// NeuroPLC — Auto-generated IEC 61131-3 SCL (DB+FB Mode)
// Graph: mlp | Target: S71500DBBackend
// Work memory: 1500KB | LUT points: 0
// Nodes: 8 | Ops: {'matmul': 4, 'standard_act': 2, 'softmax': 1, 'argmax': 1}
// Parameters in DB "NeuroPLC_MLP_Weights", inference in FB.

FUNCTION_BLOCK "NeuroPLC_Inference"
{ S7_Optimized_Access := 'FALSE' }
VERSION : 0.1

VAR_INPUT
    features : ARRAY[0..27] OF REAL;  // 28-D feature vector
END_VAR

VAR_OUTPUT
    fault_class : INT;  // 0=Normal, 1=InnerRace, 2=Ball, 3=OuterRace
    confidence : REAL;  // max softmax probability
END_VAR

VAR
    // ── Inference temporaries ──
        v1 : ARRAY[0..31] OF REAL;  // matmul output
        v2 : ARRAY[0..31] OF REAL;  // relu output
        v3 : ARRAY[0..15] OF REAL;  // matmul output
        v4 : ARRAY[0..15] OF REAL;  // relu output
        v5 : ARRAY[0..3] OF REAL;  // matmul output
        v6 : ARRAY[0..3] OF REAL;  // softmax output

    // ── Temporary variables ──
    i, o, j, lo, hi, idx, base : INT;
    sum, max_val, t_val : REAL;
END_VAR

BEGIN
    // ═══ Inference forward pass ═══
    // Parameters loaded from DB "NeuroPLC_MLP_Weights" (start values = data, not code)

        // Input: features[0..27]

        // MatMul: fc0
        v1[0] := "NeuroPLC_MLP_Weights".b1[0] + "NeuroPLC_MLP_Weights".w0[0] * features[0] + "NeuroPLC_MLP_Weights".w0[1] * features[1] + "NeuroPLC_MLP_Weights".w0[2] * features[2] + "NeuroPLC_MLP_Weights".w0[3] * features[3] + "NeuroPLC_MLP_Weights".w0[4] * features[4] + "NeuroPLC_MLP_Weights".w0[5] * features[5] + "NeuroPLC_MLP_Weights".w0[6] * features[6] + "NeuroPLC_MLP_Weights".w0[7] * features[7] + "NeuroPLC_MLP_Weights".w0[8] * features[8] + "NeuroPLC_MLP_Weights".w0[9] * features[9] + "NeuroPLC_MLP_Weights".w0[10] * features[10] + "NeuroPLC_MLP_Weights".w0[11] * features[11] + "NeuroPLC_MLP_Weights".w0[12] * features[12] + "NeuroPLC_MLP_Weights".w0[13] * features[13] + "NeuroPLC_MLP_Weights".w0[14] * features[14] + "NeuroPLC_MLP_Weights".w0[15] * features[15] + "NeuroPLC_MLP_Weights".w0[16] * features[16] + "NeuroPLC_MLP_Weights".w0[17] * features[17] + "NeuroPLC_MLP_Weights".w0[18] * features[18] + "NeuroPLC_MLP_Weights".w0[19] * features[19] + "NeuroPLC_MLP_Weights".w0[20] * features[20] + "NeuroPLC_MLP_Weights".w0[21] * features[21] + "NeuroPLC_MLP_Weights".w0[22] * features[22] + "NeuroPLC_MLP_Weights".w0[23] * features[23] + "NeuroPLC_MLP_Weights".w0[24] * features[24] + "NeuroPLC_MLP_Weights".w0[25] * features[25] + "NeuroPLC_MLP_Weights".w0[26] * features[26] + "NeuroPLC_MLP_Weights".w0[27] * features[27];
        v1[1] := "NeuroPLC_MLP_Weights".b1[1] + "NeuroPLC_MLP_Weights".w0[28] * features[0] + "NeuroPLC_MLP_Weights".w0[29] * features[1] + "NeuroPLC_MLP_Weights".w0[30] * features[2] + "NeuroPLC_MLP_Weights".w0[31] * features[3] + "NeuroPLC_MLP_Weights".w0[32] * features[4] + "NeuroPLC_MLP_Weights".w0[33] * features[5] + "NeuroPLC_MLP_Weights".w0[34] * features[6] + "NeuroPLC_MLP_Weights".w0[35] * features[7] + "NeuroPLC_MLP_Weights".w0[36] * features[8] + "NeuroPLC_MLP_Weights".w0[37] * features[9] + "NeuroPLC_MLP_Weights".w0[38] * features[10] + "NeuroPLC_MLP_Weights".w0[39] * features[11] + "NeuroPLC_MLP_Weights".w0[40] * features[12] + "NeuroPLC_MLP_Weights".w0[41] * features[13] + "NeuroPLC_MLP_Weights".w0[42] * features[14] + "NeuroPLC_MLP_Weights".w0[43] * features[15] + "NeuroPLC_MLP_Weights".w0[44] * features[16] + "NeuroPLC_MLP_Weights".w0[45] * features[17] + "NeuroPLC_MLP_Weights".w0[46] * features[18] + "NeuroPLC_MLP_Weights".w0[47] * features[19] + "NeuroPLC_MLP_Weights".w0[48] * features[20] + "NeuroPLC_MLP_Weights".w0[49] * features[21] + "NeuroPLC_MLP_Weights".w0[50] * features[22] + "NeuroPLC_MLP_Weights".w0[51] * features[23] + "NeuroPLC_MLP_Weights".w0[52] * features[24] + "NeuroPLC_MLP_Weights".w0[53] * features[25] + "NeuroPLC_MLP_Weights".w0[54] * features[26] + "NeuroPLC_MLP_Weights".w0[55] * features[27];
        v1[2] := "NeuroPLC_MLP_Weights".b1[2] + "NeuroPLC_MLP_Weights".w0[56] * features[0] + "NeuroPLC_MLP_Weights".w0[57] * features[1] + "NeuroPLC_MLP_Weights".w0[58] * features[2] + "NeuroPLC_MLP_Weights".w0[59] * features[3] + "NeuroPLC_MLP_Weights".w0[60] * features[4] + "NeuroPLC_MLP_Weights".w0[61] * features[5] + "NeuroPLC_MLP_Weights".w0[62] * features[6] + "NeuroPLC_MLP_Weights".w0[63] * features[7] + "NeuroPLC_MLP_Weights".w0[64] * features[8] + "NeuroPLC_MLP_Weights".w0[65] * features[9] + "NeuroPLC_MLP_Weights".w0[66] * features[10] + "NeuroPLC_MLP_Weights".w0[67] * features[11] + "NeuroPLC_MLP_Weights".w0[68] * features[12] + "NeuroPLC_MLP_Weights".w0[69] * features[13] + "NeuroPLC_MLP_Weights".w0[70] * features[14] + "NeuroPLC_MLP_Weights".w0[71] * features[15] + "NeuroPLC_MLP_Weights".w0[72] * features[16] + "NeuroPLC_MLP_Weights".w0[73] * features[17] + "NeuroPLC_MLP_Weights".w0[74] * features[18] + "NeuroPLC_MLP_Weights".w0[75] * features[19] + "NeuroPLC_MLP_Weights".w0[76] * features[20] + "NeuroPLC_MLP_Weights".w0[77] * features[21] + "NeuroPLC_MLP_Weights".w0[78] * features[22] + "NeuroPLC_MLP_Weights".w0[79] * features[23] + "NeuroPLC_MLP_Weights".w0[80] * features[24] + "NeuroPLC_MLP_Weights".w0[81] * features[25] + "NeuroPLC_MLP_Weights".w0[82] * features[26] + "NeuroPLC_MLP_Weights".w0[83] * features[27];
        v1[3] := "NeuroPLC_MLP_Weights".b1[3] + "NeuroPLC_MLP_Weights".w0[84] * features[0] + "NeuroPLC_MLP_Weights".w0[85] * features[1] + "NeuroPLC_MLP_Weights".w0[86] * features[2] + "NeuroPLC_MLP_Weights".w0[87] * features[3] + "NeuroPLC_MLP_Weights".w0[88] * features[4] + "NeuroPLC_MLP_Weights".w0[89] * features[5] + "NeuroPLC_MLP_Weights".w0[90] * features[6] + "NeuroPLC_MLP_Weights".w0[91] * features[7] + "NeuroPLC_MLP_Weights".w0[92] * features[8] + "NeuroPLC_MLP_Weights".w0[93] * features[9] + "NeuroPLC_MLP_Weights".w0[94] * features[10] + "NeuroPLC_MLP_Weights".w0[95] * features[11] + "NeuroPLC_MLP_Weights".w0[96] * features[12] + "NeuroPLC_MLP_Weights".w0[97] * features[13] + "NeuroPLC_MLP_Weights".w0[98] * features[14] + "NeuroPLC_MLP_Weights".w0[99] * features[15] + "NeuroPLC_MLP_Weights".w0[100] * features[16] + "NeuroPLC_MLP_Weights".w0[101] * features[17] + "NeuroPLC_MLP_Weights".w0[102] * features[18] + "NeuroPLC_MLP_Weights".w0[103] * features[19] + "NeuroPLC_MLP_Weights".w0[104] * features[20] + "NeuroPLC_MLP_Weights".w0[105] * features[21] + "NeuroPLC_MLP_Weights".w0[106] * features[22] + "NeuroPLC_MLP_Weights".w0[107] * features[23] + "NeuroPLC_MLP_Weights".w0[108] * features[24] + "NeuroPLC_MLP_Weights".w0[109] * features[25] + "NeuroPLC_MLP_Weights".w0[110] * features[26] + "NeuroPLC_MLP_Weights".w0[111] * features[27];
        v1[4] := "NeuroPLC_MLP_Weights".b1[4] + "NeuroPLC_MLP_Weights".w0[112] * features[0] + "NeuroPLC_MLP_Weights".w0[113] * features[1] + "NeuroPLC_MLP_Weights".w0[114] * features[2] + "NeuroPLC_MLP_Weights".w0[115] * features[3] + "NeuroPLC_MLP_Weights".w0[116] * features[4] + "NeuroPLC_MLP_Weights".w0[117] * features[5] + "NeuroPLC_MLP_Weights".w0[118] * features[6] + "NeuroPLC_MLP_Weights".w0[119] * features[7] + "NeuroPLC_MLP_Weights".w0[120] * features[8] + "NeuroPLC_MLP_Weights".w0[121] * features[9] + "NeuroPLC_MLP_Weights".w0[122] * features[10] + "NeuroPLC_MLP_Weights".w0[123] * features[11] + "NeuroPLC_MLP_Weights".w0[124] * features[12] + "NeuroPLC_MLP_Weights".w0[125] * features[13] + "NeuroPLC_MLP_Weights".w0[126] * features[14] + "NeuroPLC_MLP_Weights".w0[127] * features[15] + "NeuroPLC_MLP_Weights".w0[128] * features[16] + "NeuroPLC_MLP_Weights".w0[129] * features[17] + "NeuroPLC_MLP_Weights".w0[130] * features[18] + "NeuroPLC_MLP_Weights".w0[131] * features[19] + "NeuroPLC_MLP_Weights".w0[132] * features[20] + "NeuroPLC_MLP_Weights".w0[133] * features[21] + "NeuroPLC_MLP_Weights".w0[134] * features[22] + "NeuroPLC_MLP_Weights".w0[135] * features[23] + "NeuroPLC_MLP_Weights".w0[136] * features[24] + "NeuroPLC_MLP_Weights".w0[137] * features[25] + "NeuroPLC_MLP_Weights".w0[138] * features[26] + "NeuroPLC_MLP_Weights".w0[139] * features[27];
        v1[5] := "NeuroPLC_MLP_Weights".b1[5] + "NeuroPLC_MLP_Weights".w0[140] * features[0] + "NeuroPLC_MLP_Weights".w0[141] * features[1] + "NeuroPLC_MLP_Weights".w0[142] * features[2] + "NeuroPLC_MLP_Weights".w0[143] * features[3] + "NeuroPLC_MLP_Weights".w0[144] * features[4] + "NeuroPLC_MLP_Weights".w0[145] * features[5] + "NeuroPLC_MLP_Weights".w0[146] * features[6] + "NeuroPLC_MLP_Weights".w0[147] * features[7] + "NeuroPLC_MLP_Weights".w0[148] * features[8] + "NeuroPLC_MLP_Weights".w0[149] * features[9] + "NeuroPLC_MLP_Weights".w0[150] * features[10] + "NeuroPLC_MLP_Weights".w0[151] * features[11] + "NeuroPLC_MLP_Weights".w0[152] * features[12] + "NeuroPLC_MLP_Weights".w0[153] * features[13] + "NeuroPLC_MLP_Weights".w0[154] * features[14] + "NeuroPLC_MLP_Weights".w0[155] * features[15] + "NeuroPLC_MLP_Weights".w0[156] * features[16] + "NeuroPLC_MLP_Weights".w0[157] * features[17] + "NeuroPLC_MLP_Weights".w0[158] * features[18] + "NeuroPLC_MLP_Weights".w0[159] * features[19] + "NeuroPLC_MLP_Weights".w0[160] * features[20] + "NeuroPLC_MLP_Weights".w0[161] * features[21] + "NeuroPLC_MLP_Weights".w0[162] * features[22] + "NeuroPLC_MLP_Weights".w0[163] * features[23] + "NeuroPLC_MLP_Weights".w0[164] * features[24] + "NeuroPLC_MLP_Weights".w0[165] * features[25] + "NeuroPLC_MLP_Weights".w0[166] * features[26] + "NeuroPLC_MLP_Weights".w0[167] * features[27];
        v1[6] := "NeuroPLC_MLP_Weights".b1[6] + "NeuroPLC_MLP_Weights".w0[168] * features[0] + "NeuroPLC_MLP_Weights".w0[169] * features[1] + "NeuroPLC_MLP_Weights".w0[170] * features[2] + "NeuroPLC_MLP_Weights".w0[171] * features[3] + "NeuroPLC_MLP_Weights".w0[172] * features[4] + "NeuroPLC_MLP_Weights".w0[173] * features[5] + "NeuroPLC_MLP_Weights".w0[174] * features[6] + "NeuroPLC_MLP_Weights".w0[175] * features[7] + "NeuroPLC_MLP_Weights".w0[176] * features[8] + "NeuroPLC_MLP_Weights".w0[177] * features[9] + "NeuroPLC_MLP_Weights".w0[178] * features[10] + "NeuroPLC_MLP_Weights".w0[179] * features[11] + "NeuroPLC_MLP_Weights".w0[180] * features[12] + "NeuroPLC_MLP_Weights".w0[181] * features[13] + "NeuroPLC_MLP_Weights".w0[182] * features[14] + "NeuroPLC_MLP_Weights".w0[183] * features[15] + "NeuroPLC_MLP_Weights".w0[184] * features[16] + "NeuroPLC_MLP_Weights".w0[185] * features[17] + "NeuroPLC_MLP_Weights".w0[186] * features[18] + "NeuroPLC_MLP_Weights".w0[187] * features[19] + "NeuroPLC_MLP_Weights".w0[188] * features[20] + "NeuroPLC_MLP_Weights".w0[189] * features[21] + "NeuroPLC_MLP_Weights".w0[190] * features[22] + "NeuroPLC_MLP_Weights".w0[191] * features[23] + "NeuroPLC_MLP_Weights".w0[192] * features[24] + "NeuroPLC_MLP_Weights".w0[193] * features[25] + "NeuroPLC_MLP_Weights".w0[194] * features[26] + "NeuroPLC_MLP_Weights".w0[195] * features[27];
        v1[7] := "NeuroPLC_MLP_Weights".b1[7] + "NeuroPLC_MLP_Weights".w0[196] * features[0] + "NeuroPLC_MLP_Weights".w0[197] * features[1] + "NeuroPLC_MLP_Weights".w0[198] * features[2] + "NeuroPLC_MLP_Weights".w0[199] * features[3] + "NeuroPLC_MLP_Weights".w0[200] * features[4] + "NeuroPLC_MLP_Weights".w0[201] * features[5] + "NeuroPLC_MLP_Weights".w0[202] * features[6] + "NeuroPLC_MLP_Weights".w0[203] * features[7] + "NeuroPLC_MLP_Weights".w0[204] * features[8] + "NeuroPLC_MLP_Weights".w0[205] * features[9] + "NeuroPLC_MLP_Weights".w0[206] * features[10] + "NeuroPLC_MLP_Weights".w0[207] * features[11] + "NeuroPLC_MLP_Weights".w0[208] * features[12] + "NeuroPLC_MLP_Weights".w0[209] * features[13] + "NeuroPLC_MLP_Weights".w0[210] * features[14] + "NeuroPLC_MLP_Weights".w0[211] * features[15] + "NeuroPLC_MLP_Weights".w0[212] * features[16] + "NeuroPLC_MLP_Weights".w0[213] * features[17] + "NeuroPLC_MLP_Weights".w0[214] * features[18] + "NeuroPLC_MLP_Weights".w0[215] * features[19] + "NeuroPLC_MLP_Weights".w0[216] * features[20] + "NeuroPLC_MLP_Weights".w0[217] * features[21] + "NeuroPLC_MLP_Weights".w0[218] * features[22] + "NeuroPLC_MLP_Weights".w0[219] * features[23] + "NeuroPLC_MLP_Weights".w0[220] * features[24] + "NeuroPLC_MLP_Weights".w0[221] * features[25] + "NeuroPLC_MLP_Weights".w0[222] * features[26] + "NeuroPLC_MLP_Weights".w0[223] * features[27];
        v1[8] := "NeuroPLC_MLP_Weights".b1[8] + "NeuroPLC_MLP_Weights".w0[224] * features[0] + "NeuroPLC_MLP_Weights".w0[225] * features[1] + "NeuroPLC_MLP_Weights".w0[226] * features[2] + "NeuroPLC_MLP_Weights".w0[227] * features[3] + "NeuroPLC_MLP_Weights".w0[228] * features[4] + "NeuroPLC_MLP_Weights".w0[229] * features[5] + "NeuroPLC_MLP_Weights".w0[230] * features[6] + "NeuroPLC_MLP_Weights".w0[231] * features[7] + "NeuroPLC_MLP_Weights".w0[232] * features[8] + "NeuroPLC_MLP_Weights".w0[233] * features[9] + "NeuroPLC_MLP_Weights".w0[234] * features[10] + "NeuroPLC_MLP_Weights".w0[235] * features[11] + "NeuroPLC_MLP_Weights".w0[236] * features[12] + "NeuroPLC_MLP_Weights".w0[237] * features[13] + "NeuroPLC_MLP_Weights".w0[238] * features[14] + "NeuroPLC_MLP_Weights".w0[239] * features[15] + "NeuroPLC_MLP_Weights".w0[240] * features[16] + "NeuroPLC_MLP_Weights".w0[241] * features[17] + "NeuroPLC_MLP_Weights".w0[242] * features[18] + "NeuroPLC_MLP_Weights".w0[243] * features[19] + "NeuroPLC_MLP_Weights".w0[244] * features[20] + "NeuroPLC_MLP_Weights".w0[245] * features[21] + "NeuroPLC_MLP_Weights".w0[246] * features[22] + "NeuroPLC_MLP_Weights".w0[247] * features[23] + "NeuroPLC_MLP_Weights".w0[248] * features[24] + "NeuroPLC_MLP_Weights".w0[249] * features[25] + "NeuroPLC_MLP_Weights".w0[250] * features[26] + "NeuroPLC_MLP_Weights".w0[251] * features[27];
        v1[9] := "NeuroPLC_MLP_Weights".b1[9] + "NeuroPLC_MLP_Weights".w0[252] * features[0] + "NeuroPLC_MLP_Weights".w0[253] * features[1] + "NeuroPLC_MLP_Weights".w0[254] * features[2] + "NeuroPLC_MLP_Weights".w0[255] * features[3] + "NeuroPLC_MLP_Weights".w0[256] * features[4] + "NeuroPLC_MLP_Weights".w0[257] * features[5] + "NeuroPLC_MLP_Weights".w0[258] * features[6] + "NeuroPLC_MLP_Weights".w0[259] * features[7] + "NeuroPLC_MLP_Weights".w0[260] * features[8] + "NeuroPLC_MLP_Weights".w0[261] * features[9] + "NeuroPLC_MLP_Weights".w0[262] * features[10] + "NeuroPLC_MLP_Weights".w0[263] * features[11] + "NeuroPLC_MLP_Weights".w0[264] * features[12] + "NeuroPLC_MLP_Weights".w0[265] * features[13] + "NeuroPLC_MLP_Weights".w0[266] * features[14] + "NeuroPLC_MLP_Weights".w0[267] * features[15] + "NeuroPLC_MLP_Weights".w0[268] * features[16] + "NeuroPLC_MLP_Weights".w0[269] * features[17] + "NeuroPLC_MLP_Weights".w0[270] * features[18] + "NeuroPLC_MLP_Weights".w0[271] * features[19] + "NeuroPLC_MLP_Weights".w0[272] * features[20] + "NeuroPLC_MLP_Weights".w0[273] * features[21] + "NeuroPLC_MLP_Weights".w0[274] * features[22] + "NeuroPLC_MLP_Weights".w0[275] * features[23] + "NeuroPLC_MLP_Weights".w0[276] * features[24] + "NeuroPLC_MLP_Weights".w0[277] * features[25] + "NeuroPLC_MLP_Weights".w0[278] * features[26] + "NeuroPLC_MLP_Weights".w0[279] * features[27];
        v1[10] := "NeuroPLC_MLP_Weights".b1[10] + "NeuroPLC_MLP_Weights".w0[280] * features[0] + "NeuroPLC_MLP_Weights".w0[281] * features[1] + "NeuroPLC_MLP_Weights".w0[282] * features[2] + "NeuroPLC_MLP_Weights".w0[283] * features[3] + "NeuroPLC_MLP_Weights".w0[284] * features[4] + "NeuroPLC_MLP_Weights".w0[285] * features[5] + "NeuroPLC_MLP_Weights".w0[286] * features[6] + "NeuroPLC_MLP_Weights".w0[287] * features[7] + "NeuroPLC_MLP_Weights".w0[288] * features[8] + "NeuroPLC_MLP_Weights".w0[289] * features[9] + "NeuroPLC_MLP_Weights".w0[290] * features[10] + "NeuroPLC_MLP_Weights".w0[291] * features[11] + "NeuroPLC_MLP_Weights".w0[292] * features[12] + "NeuroPLC_MLP_Weights".w0[293] * features[13] + "NeuroPLC_MLP_Weights".w0[294] * features[14] + "NeuroPLC_MLP_Weights".w0[295] * features[15] + "NeuroPLC_MLP_Weights".w0[296] * features[16] + "NeuroPLC_MLP_Weights".w0[297] * features[17] + "NeuroPLC_MLP_Weights".w0[298] * features[18] + "NeuroPLC_MLP_Weights".w0[299] * features[19] + "NeuroPLC_MLP_Weights".w0[300] * features[20] + "NeuroPLC_MLP_Weights".w0[301] * features[21] + "NeuroPLC_MLP_Weights".w0[302] * features[22] + "NeuroPLC_MLP_Weights".w0[303] * features[23] + "NeuroPLC_MLP_Weights".w0[304] * features[24] + "NeuroPLC_MLP_Weights".w0[305] * features[25] + "NeuroPLC_MLP_Weights".w0[306] * features[26] + "NeuroPLC_MLP_Weights".w0[307] * features[27];
        v1[11] := "NeuroPLC_MLP_Weights".b1[11] + "NeuroPLC_MLP_Weights".w0[308] * features[0] + "NeuroPLC_MLP_Weights".w0[309] * features[1] + "NeuroPLC_MLP_Weights".w0[310] * features[2] + "NeuroPLC_MLP_Weights".w0[311] * features[3] + "NeuroPLC_MLP_Weights".w0[312] * features[4] + "NeuroPLC_MLP_Weights".w0[313] * features[5] + "NeuroPLC_MLP_Weights".w0[314] * features[6] + "NeuroPLC_MLP_Weights".w0[315] * features[7] + "NeuroPLC_MLP_Weights".w0[316] * features[8] + "NeuroPLC_MLP_Weights".w0[317] * features[9] + "NeuroPLC_MLP_Weights".w0[318] * features[10] + "NeuroPLC_MLP_Weights".w0[319] * features[11] + "NeuroPLC_MLP_Weights".w0[320] * features[12] + "NeuroPLC_MLP_Weights".w0[321] * features[13] + "NeuroPLC_MLP_Weights".w0[322] * features[14] + "NeuroPLC_MLP_Weights".w0[323] * features[15] + "NeuroPLC_MLP_Weights".w0[324] * features[16] + "NeuroPLC_MLP_Weights".w0[325] * features[17] + "NeuroPLC_MLP_Weights".w0[326] * features[18] + "NeuroPLC_MLP_Weights".w0[327] * features[19] + "NeuroPLC_MLP_Weights".w0[328] * features[20] + "NeuroPLC_MLP_Weights".w0[329] * features[21] + "NeuroPLC_MLP_Weights".w0[330] * features[22] + "NeuroPLC_MLP_Weights".w0[331] * features[23] + "NeuroPLC_MLP_Weights".w0[332] * features[24] + "NeuroPLC_MLP_Weights".w0[333] * features[25] + "NeuroPLC_MLP_Weights".w0[334] * features[26] + "NeuroPLC_MLP_Weights".w0[335] * features[27];
        v1[12] := "NeuroPLC_MLP_Weights".b1[12] + "NeuroPLC_MLP_Weights".w0[336] * features[0] + "NeuroPLC_MLP_Weights".w0[337] * features[1] + "NeuroPLC_MLP_Weights".w0[338] * features[2] + "NeuroPLC_MLP_Weights".w0[339] * features[3] + "NeuroPLC_MLP_Weights".w0[340] * features[4] + "NeuroPLC_MLP_Weights".w0[341] * features[5] + "NeuroPLC_MLP_Weights".w0[342] * features[6] + "NeuroPLC_MLP_Weights".w0[343] * features[7] + "NeuroPLC_MLP_Weights".w0[344] * features[8] + "NeuroPLC_MLP_Weights".w0[345] * features[9] + "NeuroPLC_MLP_Weights".w0[346] * features[10] + "NeuroPLC_MLP_Weights".w0[347] * features[11] + "NeuroPLC_MLP_Weights".w0[348] * features[12] + "NeuroPLC_MLP_Weights".w0[349] * features[13] + "NeuroPLC_MLP_Weights".w0[350] * features[14] + "NeuroPLC_MLP_Weights".w0[351] * features[15] + "NeuroPLC_MLP_Weights".w0[352] * features[16] + "NeuroPLC_MLP_Weights".w0[353] * features[17] + "NeuroPLC_MLP_Weights".w0[354] * features[18] + "NeuroPLC_MLP_Weights".w0[355] * features[19] + "NeuroPLC_MLP_Weights".w0[356] * features[20] + "NeuroPLC_MLP_Weights".w0[357] * features[21] + "NeuroPLC_MLP_Weights".w0[358] * features[22] + "NeuroPLC_MLP_Weights".w0[359] * features[23] + "NeuroPLC_MLP_Weights".w0[360] * features[24] + "NeuroPLC_MLP_Weights".w0[361] * features[25] + "NeuroPLC_MLP_Weights".w0[362] * features[26] + "NeuroPLC_MLP_Weights".w0[363] * features[27];
        v1[13] := "NeuroPLC_MLP_Weights".b1[13] + "NeuroPLC_MLP_Weights".w0[364] * features[0] + "NeuroPLC_MLP_Weights".w0[365] * features[1] + "NeuroPLC_MLP_Weights".w0[366] * features[2] + "NeuroPLC_MLP_Weights".w0[367] * features[3] + "NeuroPLC_MLP_Weights".w0[368] * features[4] + "NeuroPLC_MLP_Weights".w0[369] * features[5] + "NeuroPLC_MLP_Weights".w0[370] * features[6] + "NeuroPLC_MLP_Weights".w0[371] * features[7] + "NeuroPLC_MLP_Weights".w0[372] * features[8] + "NeuroPLC_MLP_Weights".w0[373] * features[9] + "NeuroPLC_MLP_Weights".w0[374] * features[10] + "NeuroPLC_MLP_Weights".w0[375] * features[11] + "NeuroPLC_MLP_Weights".w0[376] * features[12] + "NeuroPLC_MLP_Weights".w0[377] * features[13] + "NeuroPLC_MLP_Weights".w0[378] * features[14] + "NeuroPLC_MLP_Weights".w0[379] * features[15] + "NeuroPLC_MLP_Weights".w0[380] * features[16] + "NeuroPLC_MLP_Weights".w0[381] * features[17] + "NeuroPLC_MLP_Weights".w0[382] * features[18] + "NeuroPLC_MLP_Weights".w0[383] * features[19] + "NeuroPLC_MLP_Weights".w0[384] * features[20] + "NeuroPLC_MLP_Weights".w0[385] * features[21] + "NeuroPLC_MLP_Weights".w0[386] * features[22] + "NeuroPLC_MLP_Weights".w0[387] * features[23] + "NeuroPLC_MLP_Weights".w0[388] * features[24] + "NeuroPLC_MLP_Weights".w0[389] * features[25] + "NeuroPLC_MLP_Weights".w0[390] * features[26] + "NeuroPLC_MLP_Weights".w0[391] * features[27];
        v1[14] := "NeuroPLC_MLP_Weights".b1[14] + "NeuroPLC_MLP_Weights".w0[392] * features[0] + "NeuroPLC_MLP_Weights".w0[393] * features[1] + "NeuroPLC_MLP_Weights".w0[394] * features[2] + "NeuroPLC_MLP_Weights".w0[395] * features[3] + "NeuroPLC_MLP_Weights".w0[396] * features[4] + "NeuroPLC_MLP_Weights".w0[397] * features[5] + "NeuroPLC_MLP_Weights".w0[398] * features[6] + "NeuroPLC_MLP_Weights".w0[399] * features[7] + "NeuroPLC_MLP_Weights".w0[400] * features[8] + "NeuroPLC_MLP_Weights".w0[401] * features[9] + "NeuroPLC_MLP_Weights".w0[402] * features[10] + "NeuroPLC_MLP_Weights".w0[403] * features[11] + "NeuroPLC_MLP_Weights".w0[404] * features[12] + "NeuroPLC_MLP_Weights".w0[405] * features[13] + "NeuroPLC_MLP_Weights".w0[406] * features[14] + "NeuroPLC_MLP_Weights".w0[407] * features[15] + "NeuroPLC_MLP_Weights".w0[408] * features[16] + "NeuroPLC_MLP_Weights".w0[409] * features[17] + "NeuroPLC_MLP_Weights".w0[410] * features[18] + "NeuroPLC_MLP_Weights".w0[411] * features[19] + "NeuroPLC_MLP_Weights".w0[412] * features[20] + "NeuroPLC_MLP_Weights".w0[413] * features[21] + "NeuroPLC_MLP_Weights".w0[414] * features[22] + "NeuroPLC_MLP_Weights".w0[415] * features[23] + "NeuroPLC_MLP_Weights".w0[416] * features[24] + "NeuroPLC_MLP_Weights".w0[417] * features[25] + "NeuroPLC_MLP_Weights".w0[418] * features[26] + "NeuroPLC_MLP_Weights".w0[419] * features[27];
        v1[15] := "NeuroPLC_MLP_Weights".b1[15] + "NeuroPLC_MLP_Weights".w0[420] * features[0] + "NeuroPLC_MLP_Weights".w0[421] * features[1] + "NeuroPLC_MLP_Weights".w0[422] * features[2] + "NeuroPLC_MLP_Weights".w0[423] * features[3] + "NeuroPLC_MLP_Weights".w0[424] * features[4] + "NeuroPLC_MLP_Weights".w0[425] * features[5] + "NeuroPLC_MLP_Weights".w0[426] * features[6] + "NeuroPLC_MLP_Weights".w0[427] * features[7] + "NeuroPLC_MLP_Weights".w0[428] * features[8] + "NeuroPLC_MLP_Weights".w0[429] * features[9] + "NeuroPLC_MLP_Weights".w0[430] * features[10] + "NeuroPLC_MLP_Weights".w0[431] * features[11] + "NeuroPLC_MLP_Weights".w0[432] * features[12] + "NeuroPLC_MLP_Weights".w0[433] * features[13] + "NeuroPLC_MLP_Weights".w0[434] * features[14] + "NeuroPLC_MLP_Weights".w0[435] * features[15] + "NeuroPLC_MLP_Weights".w0[436] * features[16] + "NeuroPLC_MLP_Weights".w0[437] * features[17] + "NeuroPLC_MLP_Weights".w0[438] * features[18] + "NeuroPLC_MLP_Weights".w0[439] * features[19] + "NeuroPLC_MLP_Weights".w0[440] * features[20] + "NeuroPLC_MLP_Weights".w0[441] * features[21] + "NeuroPLC_MLP_Weights".w0[442] * features[22] + "NeuroPLC_MLP_Weights".w0[443] * features[23] + "NeuroPLC_MLP_Weights".w0[444] * features[24] + "NeuroPLC_MLP_Weights".w0[445] * features[25] + "NeuroPLC_MLP_Weights".w0[446] * features[26] + "NeuroPLC_MLP_Weights".w0[447] * features[27];
        v1[16] := "NeuroPLC_MLP_Weights".b1[16] + "NeuroPLC_MLP_Weights".w0[448] * features[0] + "NeuroPLC_MLP_Weights".w0[449] * features[1] + "NeuroPLC_MLP_Weights".w0[450] * features[2] + "NeuroPLC_MLP_Weights".w0[451] * features[3] + "NeuroPLC_MLP_Weights".w0[452] * features[4] + "NeuroPLC_MLP_Weights".w0[453] * features[5] + "NeuroPLC_MLP_Weights".w0[454] * features[6] + "NeuroPLC_MLP_Weights".w0[455] * features[7] + "NeuroPLC_MLP_Weights".w0[456] * features[8] + "NeuroPLC_MLP_Weights".w0[457] * features[9] + "NeuroPLC_MLP_Weights".w0[458] * features[10] + "NeuroPLC_MLP_Weights".w0[459] * features[11] + "NeuroPLC_MLP_Weights".w0[460] * features[12] + "NeuroPLC_MLP_Weights".w0[461] * features[13] + "NeuroPLC_MLP_Weights".w0[462] * features[14] + "NeuroPLC_MLP_Weights".w0[463] * features[15] + "NeuroPLC_MLP_Weights".w0[464] * features[16] + "NeuroPLC_MLP_Weights".w0[465] * features[17] + "NeuroPLC_MLP_Weights".w0[466] * features[18] + "NeuroPLC_MLP_Weights".w0[467] * features[19] + "NeuroPLC_MLP_Weights".w0[468] * features[20] + "NeuroPLC_MLP_Weights".w0[469] * features[21] + "NeuroPLC_MLP_Weights".w0[470] * features[22] + "NeuroPLC_MLP_Weights".w0[471] * features[23] + "NeuroPLC_MLP_Weights".w0[472] * features[24] + "NeuroPLC_MLP_Weights".w0[473] * features[25] + "NeuroPLC_MLP_Weights".w0[474] * features[26] + "NeuroPLC_MLP_Weights".w0[475] * features[27];
        v1[17] := "NeuroPLC_MLP_Weights".b1[17] + "NeuroPLC_MLP_Weights".w0[476] * features[0] + "NeuroPLC_MLP_Weights".w0[477] * features[1] + "NeuroPLC_MLP_Weights".w0[478] * features[2] + "NeuroPLC_MLP_Weights".w0[479] * features[3] + "NeuroPLC_MLP_Weights".w0[480] * features[4] + "NeuroPLC_MLP_Weights".w0[481] * features[5] + "NeuroPLC_MLP_Weights".w0[482] * features[6] + "NeuroPLC_MLP_Weights".w0[483] * features[7] + "NeuroPLC_MLP_Weights".w0[484] * features[8] + "NeuroPLC_MLP_Weights".w0[485] * features[9] + "NeuroPLC_MLP_Weights".w0[486] * features[10] + "NeuroPLC_MLP_Weights".w0[487] * features[11] + "NeuroPLC_MLP_Weights".w0[488] * features[12] + "NeuroPLC_MLP_Weights".w0[489] * features[13] + "NeuroPLC_MLP_Weights".w0[490] * features[14] + "NeuroPLC_MLP_Weights".w0[491] * features[15] + "NeuroPLC_MLP_Weights".w0[492] * features[16] + "NeuroPLC_MLP_Weights".w0[493] * features[17] + "NeuroPLC_MLP_Weights".w0[494] * features[18] + "NeuroPLC_MLP_Weights".w0[495] * features[19] + "NeuroPLC_MLP_Weights".w0[496] * features[20] + "NeuroPLC_MLP_Weights".w0[497] * features[21] + "NeuroPLC_MLP_Weights".w0[498] * features[22] + "NeuroPLC_MLP_Weights".w0[499] * features[23] + "NeuroPLC_MLP_Weights".w0[500] * features[24] + "NeuroPLC_MLP_Weights".w0[501] * features[25] + "NeuroPLC_MLP_Weights".w0[502] * features[26] + "NeuroPLC_MLP_Weights".w0[503] * features[27];
        v1[18] := "NeuroPLC_MLP_Weights".b1[18] + "NeuroPLC_MLP_Weights".w0[504] * features[0] + "NeuroPLC_MLP_Weights".w0[505] * features[1] + "NeuroPLC_MLP_Weights".w0[506] * features[2] + "NeuroPLC_MLP_Weights".w0[507] * features[3] + "NeuroPLC_MLP_Weights".w0[508] * features[4] + "NeuroPLC_MLP_Weights".w0[509] * features[5] + "NeuroPLC_MLP_Weights".w0[510] * features[6] + "NeuroPLC_MLP_Weights".w0[511] * features[7] + "NeuroPLC_MLP_Weights".w0[512] * features[8] + "NeuroPLC_MLP_Weights".w0[513] * features[9] + "NeuroPLC_MLP_Weights".w0[514] * features[10] + "NeuroPLC_MLP_Weights".w0[515] * features[11] + "NeuroPLC_MLP_Weights".w0[516] * features[12] + "NeuroPLC_MLP_Weights".w0[517] * features[13] + "NeuroPLC_MLP_Weights".w0[518] * features[14] + "NeuroPLC_MLP_Weights".w0[519] * features[15] + "NeuroPLC_MLP_Weights".w0[520] * features[16] + "NeuroPLC_MLP_Weights".w0[521] * features[17] + "NeuroPLC_MLP_Weights".w0[522] * features[18] + "NeuroPLC_MLP_Weights".w0[523] * features[19] + "NeuroPLC_MLP_Weights".w0[524] * features[20] + "NeuroPLC_MLP_Weights".w0[525] * features[21] + "NeuroPLC_MLP_Weights".w0[526] * features[22] + "NeuroPLC_MLP_Weights".w0[527] * features[23] + "NeuroPLC_MLP_Weights".w0[528] * features[24] + "NeuroPLC_MLP_Weights".w0[529] * features[25] + "NeuroPLC_MLP_Weights".w0[530] * features[26] + "NeuroPLC_MLP_Weights".w0[531] * features[27];
        v1[19] := "NeuroPLC_MLP_Weights".b1[19] + "NeuroPLC_MLP_Weights".w0[532] * features[0] + "NeuroPLC_MLP_Weights".w0[533] * features[1] + "NeuroPLC_MLP_Weights".w0[534] * features[2] + "NeuroPLC_MLP_Weights".w0[535] * features[3] + "NeuroPLC_MLP_Weights".w0[536] * features[4] + "NeuroPLC_MLP_Weights".w0[537] * features[5] + "NeuroPLC_MLP_Weights".w0[538] * features[6] + "NeuroPLC_MLP_Weights".w0[539] * features[7] + "NeuroPLC_MLP_Weights".w0[540] * features[8] + "NeuroPLC_MLP_Weights".w0[541] * features[9] + "NeuroPLC_MLP_Weights".w0[542] * features[10] + "NeuroPLC_MLP_Weights".w0[543] * features[11] + "NeuroPLC_MLP_Weights".w0[544] * features[12] + "NeuroPLC_MLP_Weights".w0[545] * features[13] + "NeuroPLC_MLP_Weights".w0[546] * features[14] + "NeuroPLC_MLP_Weights".w0[547] * features[15] + "NeuroPLC_MLP_Weights".w0[548] * features[16] + "NeuroPLC_MLP_Weights".w0[549] * features[17] + "NeuroPLC_MLP_Weights".w0[550] * features[18] + "NeuroPLC_MLP_Weights".w0[551] * features[19] + "NeuroPLC_MLP_Weights".w0[552] * features[20] + "NeuroPLC_MLP_Weights".w0[553] * features[21] + "NeuroPLC_MLP_Weights".w0[554] * features[22] + "NeuroPLC_MLP_Weights".w0[555] * features[23] + "NeuroPLC_MLP_Weights".w0[556] * features[24] + "NeuroPLC_MLP_Weights".w0[557] * features[25] + "NeuroPLC_MLP_Weights".w0[558] * features[26] + "NeuroPLC_MLP_Weights".w0[559] * features[27];
        v1[20] := "NeuroPLC_MLP_Weights".b1[20] + "NeuroPLC_MLP_Weights".w0[560] * features[0] + "NeuroPLC_MLP_Weights".w0[561] * features[1] + "NeuroPLC_MLP_Weights".w0[562] * features[2] + "NeuroPLC_MLP_Weights".w0[563] * features[3] + "NeuroPLC_MLP_Weights".w0[564] * features[4] + "NeuroPLC_MLP_Weights".w0[565] * features[5] + "NeuroPLC_MLP_Weights".w0[566] * features[6] + "NeuroPLC_MLP_Weights".w0[567] * features[7] + "NeuroPLC_MLP_Weights".w0[568] * features[8] + "NeuroPLC_MLP_Weights".w0[569] * features[9] + "NeuroPLC_MLP_Weights".w0[570] * features[10] + "NeuroPLC_MLP_Weights".w0[571] * features[11] + "NeuroPLC_MLP_Weights".w0[572] * features[12] + "NeuroPLC_MLP_Weights".w0[573] * features[13] + "NeuroPLC_MLP_Weights".w0[574] * features[14] + "NeuroPLC_MLP_Weights".w0[575] * features[15] + "NeuroPLC_MLP_Weights".w0[576] * features[16] + "NeuroPLC_MLP_Weights".w0[577] * features[17] + "NeuroPLC_MLP_Weights".w0[578] * features[18] + "NeuroPLC_MLP_Weights".w0[579] * features[19] + "NeuroPLC_MLP_Weights".w0[580] * features[20] + "NeuroPLC_MLP_Weights".w0[581] * features[21] + "NeuroPLC_MLP_Weights".w0[582] * features[22] + "NeuroPLC_MLP_Weights".w0[583] * features[23] + "NeuroPLC_MLP_Weights".w0[584] * features[24] + "NeuroPLC_MLP_Weights".w0[585] * features[25] + "NeuroPLC_MLP_Weights".w0[586] * features[26] + "NeuroPLC_MLP_Weights".w0[587] * features[27];
        v1[21] := "NeuroPLC_MLP_Weights".b1[21] + "NeuroPLC_MLP_Weights".w0[588] * features[0] + "NeuroPLC_MLP_Weights".w0[589] * features[1] + "NeuroPLC_MLP_Weights".w0[590] * features[2] + "NeuroPLC_MLP_Weights".w0[591] * features[3] + "NeuroPLC_MLP_Weights".w0[592] * features[4] + "NeuroPLC_MLP_Weights".w0[593] * features[5] + "NeuroPLC_MLP_Weights".w0[594] * features[6] + "NeuroPLC_MLP_Weights".w0[595] * features[7] + "NeuroPLC_MLP_Weights".w0[596] * features[8] + "NeuroPLC_MLP_Weights".w0[597] * features[9] + "NeuroPLC_MLP_Weights".w0[598] * features[10] + "NeuroPLC_MLP_Weights".w0[599] * features[11] + "NeuroPLC_MLP_Weights".w0[600] * features[12] + "NeuroPLC_MLP_Weights".w0[601] * features[13] + "NeuroPLC_MLP_Weights".w0[602] * features[14] + "NeuroPLC_MLP_Weights".w0[603] * features[15] + "NeuroPLC_MLP_Weights".w0[604] * features[16] + "NeuroPLC_MLP_Weights".w0[605] * features[17] + "NeuroPLC_MLP_Weights".w0[606] * features[18] + "NeuroPLC_MLP_Weights".w0[607] * features[19] + "NeuroPLC_MLP_Weights".w0[608] * features[20] + "NeuroPLC_MLP_Weights".w0[609] * features[21] + "NeuroPLC_MLP_Weights".w0[610] * features[22] + "NeuroPLC_MLP_Weights".w0[611] * features[23] + "NeuroPLC_MLP_Weights".w0[612] * features[24] + "NeuroPLC_MLP_Weights".w0[613] * features[25] + "NeuroPLC_MLP_Weights".w0[614] * features[26] + "NeuroPLC_MLP_Weights".w0[615] * features[27];
        v1[22] := "NeuroPLC_MLP_Weights".b1[22] + "NeuroPLC_MLP_Weights".w0[616] * features[0] + "NeuroPLC_MLP_Weights".w0[617] * features[1] + "NeuroPLC_MLP_Weights".w0[618] * features[2] + "NeuroPLC_MLP_Weights".w0[619] * features[3] + "NeuroPLC_MLP_Weights".w0[620] * features[4] + "NeuroPLC_MLP_Weights".w0[621] * features[5] + "NeuroPLC_MLP_Weights".w0[622] * features[6] + "NeuroPLC_MLP_Weights".w0[623] * features[7] + "NeuroPLC_MLP_Weights".w0[624] * features[8] + "NeuroPLC_MLP_Weights".w0[625] * features[9] + "NeuroPLC_MLP_Weights".w0[626] * features[10] + "NeuroPLC_MLP_Weights".w0[627] * features[11] + "NeuroPLC_MLP_Weights".w0[628] * features[12] + "NeuroPLC_MLP_Weights".w0[629] * features[13] + "NeuroPLC_MLP_Weights".w0[630] * features[14] + "NeuroPLC_MLP_Weights".w0[631] * features[15] + "NeuroPLC_MLP_Weights".w0[632] * features[16] + "NeuroPLC_MLP_Weights".w0[633] * features[17] + "NeuroPLC_MLP_Weights".w0[634] * features[18] + "NeuroPLC_MLP_Weights".w0[635] * features[19] + "NeuroPLC_MLP_Weights".w0[636] * features[20] + "NeuroPLC_MLP_Weights".w0[637] * features[21] + "NeuroPLC_MLP_Weights".w0[638] * features[22] + "NeuroPLC_MLP_Weights".w0[639] * features[23] + "NeuroPLC_MLP_Weights".w0[640] * features[24] + "NeuroPLC_MLP_Weights".w0[641] * features[25] + "NeuroPLC_MLP_Weights".w0[642] * features[26] + "NeuroPLC_MLP_Weights".w0[643] * features[27];
        v1[23] := "NeuroPLC_MLP_Weights".b1[23] + "NeuroPLC_MLP_Weights".w0[644] * features[0] + "NeuroPLC_MLP_Weights".w0[645] * features[1] + "NeuroPLC_MLP_Weights".w0[646] * features[2] + "NeuroPLC_MLP_Weights".w0[647] * features[3] + "NeuroPLC_MLP_Weights".w0[648] * features[4] + "NeuroPLC_MLP_Weights".w0[649] * features[5] + "NeuroPLC_MLP_Weights".w0[650] * features[6] + "NeuroPLC_MLP_Weights".w0[651] * features[7] + "NeuroPLC_MLP_Weights".w0[652] * features[8] + "NeuroPLC_MLP_Weights".w0[653] * features[9] + "NeuroPLC_MLP_Weights".w0[654] * features[10] + "NeuroPLC_MLP_Weights".w0[655] * features[11] + "NeuroPLC_MLP_Weights".w0[656] * features[12] + "NeuroPLC_MLP_Weights".w0[657] * features[13] + "NeuroPLC_MLP_Weights".w0[658] * features[14] + "NeuroPLC_MLP_Weights".w0[659] * features[15] + "NeuroPLC_MLP_Weights".w0[660] * features[16] + "NeuroPLC_MLP_Weights".w0[661] * features[17] + "NeuroPLC_MLP_Weights".w0[662] * features[18] + "NeuroPLC_MLP_Weights".w0[663] * features[19] + "NeuroPLC_MLP_Weights".w0[664] * features[20] + "NeuroPLC_MLP_Weights".w0[665] * features[21] + "NeuroPLC_MLP_Weights".w0[666] * features[22] + "NeuroPLC_MLP_Weights".w0[667] * features[23] + "NeuroPLC_MLP_Weights".w0[668] * features[24] + "NeuroPLC_MLP_Weights".w0[669] * features[25] + "NeuroPLC_MLP_Weights".w0[670] * features[26] + "NeuroPLC_MLP_Weights".w0[671] * features[27];
        v1[24] := "NeuroPLC_MLP_Weights".b1[24] + "NeuroPLC_MLP_Weights".w0[672] * features[0] + "NeuroPLC_MLP_Weights".w0[673] * features[1] + "NeuroPLC_MLP_Weights".w0[674] * features[2] + "NeuroPLC_MLP_Weights".w0[675] * features[3] + "NeuroPLC_MLP_Weights".w0[676] * features[4] + "NeuroPLC_MLP_Weights".w0[677] * features[5] + "NeuroPLC_MLP_Weights".w0[678] * features[6] + "NeuroPLC_MLP_Weights".w0[679] * features[7] + "NeuroPLC_MLP_Weights".w0[680] * features[8] + "NeuroPLC_MLP_Weights".w0[681] * features[9] + "NeuroPLC_MLP_Weights".w0[682] * features[10] + "NeuroPLC_MLP_Weights".w0[683] * features[11] + "NeuroPLC_MLP_Weights".w0[684] * features[12] + "NeuroPLC_MLP_Weights".w0[685] * features[13] + "NeuroPLC_MLP_Weights".w0[686] * features[14] + "NeuroPLC_MLP_Weights".w0[687] * features[15] + "NeuroPLC_MLP_Weights".w0[688] * features[16] + "NeuroPLC_MLP_Weights".w0[689] * features[17] + "NeuroPLC_MLP_Weights".w0[690] * features[18] + "NeuroPLC_MLP_Weights".w0[691] * features[19] + "NeuroPLC_MLP_Weights".w0[692] * features[20] + "NeuroPLC_MLP_Weights".w0[693] * features[21] + "NeuroPLC_MLP_Weights".w0[694] * features[22] + "NeuroPLC_MLP_Weights".w0[695] * features[23] + "NeuroPLC_MLP_Weights".w0[696] * features[24] + "NeuroPLC_MLP_Weights".w0[697] * features[25] + "NeuroPLC_MLP_Weights".w0[698] * features[26] + "NeuroPLC_MLP_Weights".w0[699] * features[27];
        v1[25] := "NeuroPLC_MLP_Weights".b1[25] + "NeuroPLC_MLP_Weights".w0[700] * features[0] + "NeuroPLC_MLP_Weights".w0[701] * features[1] + "NeuroPLC_MLP_Weights".w0[702] * features[2] + "NeuroPLC_MLP_Weights".w0[703] * features[3] + "NeuroPLC_MLP_Weights".w0[704] * features[4] + "NeuroPLC_MLP_Weights".w0[705] * features[5] + "NeuroPLC_MLP_Weights".w0[706] * features[6] + "NeuroPLC_MLP_Weights".w0[707] * features[7] + "NeuroPLC_MLP_Weights".w0[708] * features[8] + "NeuroPLC_MLP_Weights".w0[709] * features[9] + "NeuroPLC_MLP_Weights".w0[710] * features[10] + "NeuroPLC_MLP_Weights".w0[711] * features[11] + "NeuroPLC_MLP_Weights".w0[712] * features[12] + "NeuroPLC_MLP_Weights".w0[713] * features[13] + "NeuroPLC_MLP_Weights".w0[714] * features[14] + "NeuroPLC_MLP_Weights".w0[715] * features[15] + "NeuroPLC_MLP_Weights".w0[716] * features[16] + "NeuroPLC_MLP_Weights".w0[717] * features[17] + "NeuroPLC_MLP_Weights".w0[718] * features[18] + "NeuroPLC_MLP_Weights".w0[719] * features[19] + "NeuroPLC_MLP_Weights".w0[720] * features[20] + "NeuroPLC_MLP_Weights".w0[721] * features[21] + "NeuroPLC_MLP_Weights".w0[722] * features[22] + "NeuroPLC_MLP_Weights".w0[723] * features[23] + "NeuroPLC_MLP_Weights".w0[724] * features[24] + "NeuroPLC_MLP_Weights".w0[725] * features[25] + "NeuroPLC_MLP_Weights".w0[726] * features[26] + "NeuroPLC_MLP_Weights".w0[727] * features[27];
        v1[26] := "NeuroPLC_MLP_Weights".b1[26] + "NeuroPLC_MLP_Weights".w0[728] * features[0] + "NeuroPLC_MLP_Weights".w0[729] * features[1] + "NeuroPLC_MLP_Weights".w0[730] * features[2] + "NeuroPLC_MLP_Weights".w0[731] * features[3] + "NeuroPLC_MLP_Weights".w0[732] * features[4] + "NeuroPLC_MLP_Weights".w0[733] * features[5] + "NeuroPLC_MLP_Weights".w0[734] * features[6] + "NeuroPLC_MLP_Weights".w0[735] * features[7] + "NeuroPLC_MLP_Weights".w0[736] * features[8] + "NeuroPLC_MLP_Weights".w0[737] * features[9] + "NeuroPLC_MLP_Weights".w0[738] * features[10] + "NeuroPLC_MLP_Weights".w0[739] * features[11] + "NeuroPLC_MLP_Weights".w0[740] * features[12] + "NeuroPLC_MLP_Weights".w0[741] * features[13] + "NeuroPLC_MLP_Weights".w0[742] * features[14] + "NeuroPLC_MLP_Weights".w0[743] * features[15] + "NeuroPLC_MLP_Weights".w0[744] * features[16] + "NeuroPLC_MLP_Weights".w0[745] * features[17] + "NeuroPLC_MLP_Weights".w0[746] * features[18] + "NeuroPLC_MLP_Weights".w0[747] * features[19] + "NeuroPLC_MLP_Weights".w0[748] * features[20] + "NeuroPLC_MLP_Weights".w0[749] * features[21] + "NeuroPLC_MLP_Weights".w0[750] * features[22] + "NeuroPLC_MLP_Weights".w0[751] * features[23] + "NeuroPLC_MLP_Weights".w0[752] * features[24] + "NeuroPLC_MLP_Weights".w0[753] * features[25] + "NeuroPLC_MLP_Weights".w0[754] * features[26] + "NeuroPLC_MLP_Weights".w0[755] * features[27];
        v1[27] := "NeuroPLC_MLP_Weights".b1[27] + "NeuroPLC_MLP_Weights".w0[756] * features[0] + "NeuroPLC_MLP_Weights".w0[757] * features[1] + "NeuroPLC_MLP_Weights".w0[758] * features[2] + "NeuroPLC_MLP_Weights".w0[759] * features[3] + "NeuroPLC_MLP_Weights".w0[760] * features[4] + "NeuroPLC_MLP_Weights".w0[761] * features[5] + "NeuroPLC_MLP_Weights".w0[762] * features[6] + "NeuroPLC_MLP_Weights".w0[763] * features[7] + "NeuroPLC_MLP_Weights".w0[764] * features[8] + "NeuroPLC_MLP_Weights".w0[765] * features[9] + "NeuroPLC_MLP_Weights".w0[766] * features[10] + "NeuroPLC_MLP_Weights".w0[767] * features[11] + "NeuroPLC_MLP_Weights".w0[768] * features[12] + "NeuroPLC_MLP_Weights".w0[769] * features[13] + "NeuroPLC_MLP_Weights".w0[770] * features[14] + "NeuroPLC_MLP_Weights".w0[771] * features[15] + "NeuroPLC_MLP_Weights".w0[772] * features[16] + "NeuroPLC_MLP_Weights".w0[773] * features[17] + "NeuroPLC_MLP_Weights".w0[774] * features[18] + "NeuroPLC_MLP_Weights".w0[775] * features[19] + "NeuroPLC_MLP_Weights".w0[776] * features[20] + "NeuroPLC_MLP_Weights".w0[777] * features[21] + "NeuroPLC_MLP_Weights".w0[778] * features[22] + "NeuroPLC_MLP_Weights".w0[779] * features[23] + "NeuroPLC_MLP_Weights".w0[780] * features[24] + "NeuroPLC_MLP_Weights".w0[781] * features[25] + "NeuroPLC_MLP_Weights".w0[782] * features[26] + "NeuroPLC_MLP_Weights".w0[783] * features[27];
        v1[28] := "NeuroPLC_MLP_Weights".b1[28] + "NeuroPLC_MLP_Weights".w0[784] * features[0] + "NeuroPLC_MLP_Weights".w0[785] * features[1] + "NeuroPLC_MLP_Weights".w0[786] * features[2] + "NeuroPLC_MLP_Weights".w0[787] * features[3] + "NeuroPLC_MLP_Weights".w0[788] * features[4] + "NeuroPLC_MLP_Weights".w0[789] * features[5] + "NeuroPLC_MLP_Weights".w0[790] * features[6] + "NeuroPLC_MLP_Weights".w0[791] * features[7] + "NeuroPLC_MLP_Weights".w0[792] * features[8] + "NeuroPLC_MLP_Weights".w0[793] * features[9] + "NeuroPLC_MLP_Weights".w0[794] * features[10] + "NeuroPLC_MLP_Weights".w0[795] * features[11] + "NeuroPLC_MLP_Weights".w0[796] * features[12] + "NeuroPLC_MLP_Weights".w0[797] * features[13] + "NeuroPLC_MLP_Weights".w0[798] * features[14] + "NeuroPLC_MLP_Weights".w0[799] * features[15] + "NeuroPLC_MLP_Weights".w0[800] * features[16] + "NeuroPLC_MLP_Weights".w0[801] * features[17] + "NeuroPLC_MLP_Weights".w0[802] * features[18] + "NeuroPLC_MLP_Weights".w0[803] * features[19] + "NeuroPLC_MLP_Weights".w0[804] * features[20] + "NeuroPLC_MLP_Weights".w0[805] * features[21] + "NeuroPLC_MLP_Weights".w0[806] * features[22] + "NeuroPLC_MLP_Weights".w0[807] * features[23] + "NeuroPLC_MLP_Weights".w0[808] * features[24] + "NeuroPLC_MLP_Weights".w0[809] * features[25] + "NeuroPLC_MLP_Weights".w0[810] * features[26] + "NeuroPLC_MLP_Weights".w0[811] * features[27];
        v1[29] := "NeuroPLC_MLP_Weights".b1[29] + "NeuroPLC_MLP_Weights".w0[812] * features[0] + "NeuroPLC_MLP_Weights".w0[813] * features[1] + "NeuroPLC_MLP_Weights".w0[814] * features[2] + "NeuroPLC_MLP_Weights".w0[815] * features[3] + "NeuroPLC_MLP_Weights".w0[816] * features[4] + "NeuroPLC_MLP_Weights".w0[817] * features[5] + "NeuroPLC_MLP_Weights".w0[818] * features[6] + "NeuroPLC_MLP_Weights".w0[819] * features[7] + "NeuroPLC_MLP_Weights".w0[820] * features[8] + "NeuroPLC_MLP_Weights".w0[821] * features[9] + "NeuroPLC_MLP_Weights".w0[822] * features[10] + "NeuroPLC_MLP_Weights".w0[823] * features[11] + "NeuroPLC_MLP_Weights".w0[824] * features[12] + "NeuroPLC_MLP_Weights".w0[825] * features[13] + "NeuroPLC_MLP_Weights".w0[826] * features[14] + "NeuroPLC_MLP_Weights".w0[827] * features[15] + "NeuroPLC_MLP_Weights".w0[828] * features[16] + "NeuroPLC_MLP_Weights".w0[829] * features[17] + "NeuroPLC_MLP_Weights".w0[830] * features[18] + "NeuroPLC_MLP_Weights".w0[831] * features[19] + "NeuroPLC_MLP_Weights".w0[832] * features[20] + "NeuroPLC_MLP_Weights".w0[833] * features[21] + "NeuroPLC_MLP_Weights".w0[834] * features[22] + "NeuroPLC_MLP_Weights".w0[835] * features[23] + "NeuroPLC_MLP_Weights".w0[836] * features[24] + "NeuroPLC_MLP_Weights".w0[837] * features[25] + "NeuroPLC_MLP_Weights".w0[838] * features[26] + "NeuroPLC_MLP_Weights".w0[839] * features[27];
        v1[30] := "NeuroPLC_MLP_Weights".b1[30] + "NeuroPLC_MLP_Weights".w0[840] * features[0] + "NeuroPLC_MLP_Weights".w0[841] * features[1] + "NeuroPLC_MLP_Weights".w0[842] * features[2] + "NeuroPLC_MLP_Weights".w0[843] * features[3] + "NeuroPLC_MLP_Weights".w0[844] * features[4] + "NeuroPLC_MLP_Weights".w0[845] * features[5] + "NeuroPLC_MLP_Weights".w0[846] * features[6] + "NeuroPLC_MLP_Weights".w0[847] * features[7] + "NeuroPLC_MLP_Weights".w0[848] * features[8] + "NeuroPLC_MLP_Weights".w0[849] * features[9] + "NeuroPLC_MLP_Weights".w0[850] * features[10] + "NeuroPLC_MLP_Weights".w0[851] * features[11] + "NeuroPLC_MLP_Weights".w0[852] * features[12] + "NeuroPLC_MLP_Weights".w0[853] * features[13] + "NeuroPLC_MLP_Weights".w0[854] * features[14] + "NeuroPLC_MLP_Weights".w0[855] * features[15] + "NeuroPLC_MLP_Weights".w0[856] * features[16] + "NeuroPLC_MLP_Weights".w0[857] * features[17] + "NeuroPLC_MLP_Weights".w0[858] * features[18] + "NeuroPLC_MLP_Weights".w0[859] * features[19] + "NeuroPLC_MLP_Weights".w0[860] * features[20] + "NeuroPLC_MLP_Weights".w0[861] * features[21] + "NeuroPLC_MLP_Weights".w0[862] * features[22] + "NeuroPLC_MLP_Weights".w0[863] * features[23] + "NeuroPLC_MLP_Weights".w0[864] * features[24] + "NeuroPLC_MLP_Weights".w0[865] * features[25] + "NeuroPLC_MLP_Weights".w0[866] * features[26] + "NeuroPLC_MLP_Weights".w0[867] * features[27];
        v1[31] := "NeuroPLC_MLP_Weights".b1[31] + "NeuroPLC_MLP_Weights".w0[868] * features[0] + "NeuroPLC_MLP_Weights".w0[869] * features[1] + "NeuroPLC_MLP_Weights".w0[870] * features[2] + "NeuroPLC_MLP_Weights".w0[871] * features[3] + "NeuroPLC_MLP_Weights".w0[872] * features[4] + "NeuroPLC_MLP_Weights".w0[873] * features[5] + "NeuroPLC_MLP_Weights".w0[874] * features[6] + "NeuroPLC_MLP_Weights".w0[875] * features[7] + "NeuroPLC_MLP_Weights".w0[876] * features[8] + "NeuroPLC_MLP_Weights".w0[877] * features[9] + "NeuroPLC_MLP_Weights".w0[878] * features[10] + "NeuroPLC_MLP_Weights".w0[879] * features[11] + "NeuroPLC_MLP_Weights".w0[880] * features[12] + "NeuroPLC_MLP_Weights".w0[881] * features[13] + "NeuroPLC_MLP_Weights".w0[882] * features[14] + "NeuroPLC_MLP_Weights".w0[883] * features[15] + "NeuroPLC_MLP_Weights".w0[884] * features[16] + "NeuroPLC_MLP_Weights".w0[885] * features[17] + "NeuroPLC_MLP_Weights".w0[886] * features[18] + "NeuroPLC_MLP_Weights".w0[887] * features[19] + "NeuroPLC_MLP_Weights".w0[888] * features[20] + "NeuroPLC_MLP_Weights".w0[889] * features[21] + "NeuroPLC_MLP_Weights".w0[890] * features[22] + "NeuroPLC_MLP_Weights".w0[891] * features[23] + "NeuroPLC_MLP_Weights".w0[892] * features[24] + "NeuroPLC_MLP_Weights".w0[893] * features[25] + "NeuroPLC_MLP_Weights".w0[894] * features[26] + "NeuroPLC_MLP_Weights".w0[895] * features[27];

        // StandardAct: relu
        FOR i := 0 TO 31 DO
            IF v1[i] < 0.0 THEN
                v2[i] := 0.0;
            ELSE
                v2[i] := v1[i];
            END_IF;
        END_FOR;

        // MatMul: fc1
        v3[0] := "NeuroPLC_MLP_Weights".b3[0] + "NeuroPLC_MLP_Weights".w2[0] * v2[0] + "NeuroPLC_MLP_Weights".w2[1] * v2[1] + "NeuroPLC_MLP_Weights".w2[2] * v2[2] + "NeuroPLC_MLP_Weights".w2[3] * v2[3] + "NeuroPLC_MLP_Weights".w2[4] * v2[4] + "NeuroPLC_MLP_Weights".w2[5] * v2[5] + "NeuroPLC_MLP_Weights".w2[6] * v2[6] + "NeuroPLC_MLP_Weights".w2[7] * v2[7] + "NeuroPLC_MLP_Weights".w2[8] * v2[8] + "NeuroPLC_MLP_Weights".w2[9] * v2[9] + "NeuroPLC_MLP_Weights".w2[10] * v2[10] + "NeuroPLC_MLP_Weights".w2[11] * v2[11] + "NeuroPLC_MLP_Weights".w2[12] * v2[12] + "NeuroPLC_MLP_Weights".w2[13] * v2[13] + "NeuroPLC_MLP_Weights".w2[14] * v2[14] + "NeuroPLC_MLP_Weights".w2[15] * v2[15] + "NeuroPLC_MLP_Weights".w2[16] * v2[16] + "NeuroPLC_MLP_Weights".w2[17] * v2[17] + "NeuroPLC_MLP_Weights".w2[18] * v2[18] + "NeuroPLC_MLP_Weights".w2[19] * v2[19] + "NeuroPLC_MLP_Weights".w2[20] * v2[20] + "NeuroPLC_MLP_Weights".w2[21] * v2[21] + "NeuroPLC_MLP_Weights".w2[22] * v2[22] + "NeuroPLC_MLP_Weights".w2[23] * v2[23] + "NeuroPLC_MLP_Weights".w2[24] * v2[24] + "NeuroPLC_MLP_Weights".w2[25] * v2[25] + "NeuroPLC_MLP_Weights".w2[26] * v2[26] + "NeuroPLC_MLP_Weights".w2[27] * v2[27] + "NeuroPLC_MLP_Weights".w2[28] * v2[28] + "NeuroPLC_MLP_Weights".w2[29] * v2[29] + "NeuroPLC_MLP_Weights".w2[30] * v2[30] + "NeuroPLC_MLP_Weights".w2[31] * v2[31];
        v3[1] := "NeuroPLC_MLP_Weights".b3[1] + "NeuroPLC_MLP_Weights".w2[32] * v2[0] + "NeuroPLC_MLP_Weights".w2[33] * v2[1] + "NeuroPLC_MLP_Weights".w2[34] * v2[2] + "NeuroPLC_MLP_Weights".w2[35] * v2[3] + "NeuroPLC_MLP_Weights".w2[36] * v2[4] + "NeuroPLC_MLP_Weights".w2[37] * v2[5] + "NeuroPLC_MLP_Weights".w2[38] * v2[6] + "NeuroPLC_MLP_Weights".w2[39] * v2[7] + "NeuroPLC_MLP_Weights".w2[40] * v2[8] + "NeuroPLC_MLP_Weights".w2[41] * v2[9] + "NeuroPLC_MLP_Weights".w2[42] * v2[10] + "NeuroPLC_MLP_Weights".w2[43] * v2[11] + "NeuroPLC_MLP_Weights".w2[44] * v2[12] + "NeuroPLC_MLP_Weights".w2[45] * v2[13] + "NeuroPLC_MLP_Weights".w2[46] * v2[14] + "NeuroPLC_MLP_Weights".w2[47] * v2[15] + "NeuroPLC_MLP_Weights".w2[48] * v2[16] + "NeuroPLC_MLP_Weights".w2[49] * v2[17] + "NeuroPLC_MLP_Weights".w2[50] * v2[18] + "NeuroPLC_MLP_Weights".w2[51] * v2[19] + "NeuroPLC_MLP_Weights".w2[52] * v2[20] + "NeuroPLC_MLP_Weights".w2[53] * v2[21] + "NeuroPLC_MLP_Weights".w2[54] * v2[22] + "NeuroPLC_MLP_Weights".w2[55] * v2[23] + "NeuroPLC_MLP_Weights".w2[56] * v2[24] + "NeuroPLC_MLP_Weights".w2[57] * v2[25] + "NeuroPLC_MLP_Weights".w2[58] * v2[26] + "NeuroPLC_MLP_Weights".w2[59] * v2[27] + "NeuroPLC_MLP_Weights".w2[60] * v2[28] + "NeuroPLC_MLP_Weights".w2[61] * v2[29] + "NeuroPLC_MLP_Weights".w2[62] * v2[30] + "NeuroPLC_MLP_Weights".w2[63] * v2[31];
        v3[2] := "NeuroPLC_MLP_Weights".b3[2] + "NeuroPLC_MLP_Weights".w2[64] * v2[0] + "NeuroPLC_MLP_Weights".w2[65] * v2[1] + "NeuroPLC_MLP_Weights".w2[66] * v2[2] + "NeuroPLC_MLP_Weights".w2[67] * v2[3] + "NeuroPLC_MLP_Weights".w2[68] * v2[4] + "NeuroPLC_MLP_Weights".w2[69] * v2[5] + "NeuroPLC_MLP_Weights".w2[70] * v2[6] + "NeuroPLC_MLP_Weights".w2[71] * v2[7] + "NeuroPLC_MLP_Weights".w2[72] * v2[8] + "NeuroPLC_MLP_Weights".w2[73] * v2[9] + "NeuroPLC_MLP_Weights".w2[74] * v2[10] + "NeuroPLC_MLP_Weights".w2[75] * v2[11] + "NeuroPLC_MLP_Weights".w2[76] * v2[12] + "NeuroPLC_MLP_Weights".w2[77] * v2[13] + "NeuroPLC_MLP_Weights".w2[78] * v2[14] + "NeuroPLC_MLP_Weights".w2[79] * v2[15] + "NeuroPLC_MLP_Weights".w2[80] * v2[16] + "NeuroPLC_MLP_Weights".w2[81] * v2[17] + "NeuroPLC_MLP_Weights".w2[82] * v2[18] + "NeuroPLC_MLP_Weights".w2[83] * v2[19] + "NeuroPLC_MLP_Weights".w2[84] * v2[20] + "NeuroPLC_MLP_Weights".w2[85] * v2[21] + "NeuroPLC_MLP_Weights".w2[86] * v2[22] + "NeuroPLC_MLP_Weights".w2[87] * v2[23] + "NeuroPLC_MLP_Weights".w2[88] * v2[24] + "NeuroPLC_MLP_Weights".w2[89] * v2[25] + "NeuroPLC_MLP_Weights".w2[90] * v2[26] + "NeuroPLC_MLP_Weights".w2[91] * v2[27] + "NeuroPLC_MLP_Weights".w2[92] * v2[28] + "NeuroPLC_MLP_Weights".w2[93] * v2[29] + "NeuroPLC_MLP_Weights".w2[94] * v2[30] + "NeuroPLC_MLP_Weights".w2[95] * v2[31];
        v3[3] := "NeuroPLC_MLP_Weights".b3[3] + "NeuroPLC_MLP_Weights".w2[96] * v2[0] + "NeuroPLC_MLP_Weights".w2[97] * v2[1] + "NeuroPLC_MLP_Weights".w2[98] * v2[2] + "NeuroPLC_MLP_Weights".w2[99] * v2[3] + "NeuroPLC_MLP_Weights".w2[100] * v2[4] + "NeuroPLC_MLP_Weights".w2[101] * v2[5] + "NeuroPLC_MLP_Weights".w2[102] * v2[6] + "NeuroPLC_MLP_Weights".w2[103] * v2[7] + "NeuroPLC_MLP_Weights".w2[104] * v2[8] + "NeuroPLC_MLP_Weights".w2[105] * v2[9] + "NeuroPLC_MLP_Weights".w2[106] * v2[10] + "NeuroPLC_MLP_Weights".w2[107] * v2[11] + "NeuroPLC_MLP_Weights".w2[108] * v2[12] + "NeuroPLC_MLP_Weights".w2[109] * v2[13] + "NeuroPLC_MLP_Weights".w2[110] * v2[14] + "NeuroPLC_MLP_Weights".w2[111] * v2[15] + "NeuroPLC_MLP_Weights".w2[112] * v2[16] + "NeuroPLC_MLP_Weights".w2[113] * v2[17] + "NeuroPLC_MLP_Weights".w2[114] * v2[18] + "NeuroPLC_MLP_Weights".w2[115] * v2[19] + "NeuroPLC_MLP_Weights".w2[116] * v2[20] + "NeuroPLC_MLP_Weights".w2[117] * v2[21] + "NeuroPLC_MLP_Weights".w2[118] * v2[22] + "NeuroPLC_MLP_Weights".w2[119] * v2[23] + "NeuroPLC_MLP_Weights".w2[120] * v2[24] + "NeuroPLC_MLP_Weights".w2[121] * v2[25] + "NeuroPLC_MLP_Weights".w2[122] * v2[26] + "NeuroPLC_MLP_Weights".w2[123] * v2[27] + "NeuroPLC_MLP_Weights".w2[124] * v2[28] + "NeuroPLC_MLP_Weights".w2[125] * v2[29] + "NeuroPLC_MLP_Weights".w2[126] * v2[30] + "NeuroPLC_MLP_Weights".w2[127] * v2[31];
        v3[4] := "NeuroPLC_MLP_Weights".b3[4] + "NeuroPLC_MLP_Weights".w2[128] * v2[0] + "NeuroPLC_MLP_Weights".w2[129] * v2[1] + "NeuroPLC_MLP_Weights".w2[130] * v2[2] + "NeuroPLC_MLP_Weights".w2[131] * v2[3] + "NeuroPLC_MLP_Weights".w2[132] * v2[4] + "NeuroPLC_MLP_Weights".w2[133] * v2[5] + "NeuroPLC_MLP_Weights".w2[134] * v2[6] + "NeuroPLC_MLP_Weights".w2[135] * v2[7] + "NeuroPLC_MLP_Weights".w2[136] * v2[8] + "NeuroPLC_MLP_Weights".w2[137] * v2[9] + "NeuroPLC_MLP_Weights".w2[138] * v2[10] + "NeuroPLC_MLP_Weights".w2[139] * v2[11] + "NeuroPLC_MLP_Weights".w2[140] * v2[12] + "NeuroPLC_MLP_Weights".w2[141] * v2[13] + "NeuroPLC_MLP_Weights".w2[142] * v2[14] + "NeuroPLC_MLP_Weights".w2[143] * v2[15] + "NeuroPLC_MLP_Weights".w2[144] * v2[16] + "NeuroPLC_MLP_Weights".w2[145] * v2[17] + "NeuroPLC_MLP_Weights".w2[146] * v2[18] + "NeuroPLC_MLP_Weights".w2[147] * v2[19] + "NeuroPLC_MLP_Weights".w2[148] * v2[20] + "NeuroPLC_MLP_Weights".w2[149] * v2[21] + "NeuroPLC_MLP_Weights".w2[150] * v2[22] + "NeuroPLC_MLP_Weights".w2[151] * v2[23] + "NeuroPLC_MLP_Weights".w2[152] * v2[24] + "NeuroPLC_MLP_Weights".w2[153] * v2[25] + "NeuroPLC_MLP_Weights".w2[154] * v2[26] + "NeuroPLC_MLP_Weights".w2[155] * v2[27] + "NeuroPLC_MLP_Weights".w2[156] * v2[28] + "NeuroPLC_MLP_Weights".w2[157] * v2[29] + "NeuroPLC_MLP_Weights".w2[158] * v2[30] + "NeuroPLC_MLP_Weights".w2[159] * v2[31];
        v3[5] := "NeuroPLC_MLP_Weights".b3[5] + "NeuroPLC_MLP_Weights".w2[160] * v2[0] + "NeuroPLC_MLP_Weights".w2[161] * v2[1] + "NeuroPLC_MLP_Weights".w2[162] * v2[2] + "NeuroPLC_MLP_Weights".w2[163] * v2[3] + "NeuroPLC_MLP_Weights".w2[164] * v2[4] + "NeuroPLC_MLP_Weights".w2[165] * v2[5] + "NeuroPLC_MLP_Weights".w2[166] * v2[6] + "NeuroPLC_MLP_Weights".w2[167] * v2[7] + "NeuroPLC_MLP_Weights".w2[168] * v2[8] + "NeuroPLC_MLP_Weights".w2[169] * v2[9] + "NeuroPLC_MLP_Weights".w2[170] * v2[10] + "NeuroPLC_MLP_Weights".w2[171] * v2[11] + "NeuroPLC_MLP_Weights".w2[172] * v2[12] + "NeuroPLC_MLP_Weights".w2[173] * v2[13] + "NeuroPLC_MLP_Weights".w2[174] * v2[14] + "NeuroPLC_MLP_Weights".w2[175] * v2[15] + "NeuroPLC_MLP_Weights".w2[176] * v2[16] + "NeuroPLC_MLP_Weights".w2[177] * v2[17] + "NeuroPLC_MLP_Weights".w2[178] * v2[18] + "NeuroPLC_MLP_Weights".w2[179] * v2[19] + "NeuroPLC_MLP_Weights".w2[180] * v2[20] + "NeuroPLC_MLP_Weights".w2[181] * v2[21] + "NeuroPLC_MLP_Weights".w2[182] * v2[22] + "NeuroPLC_MLP_Weights".w2[183] * v2[23] + "NeuroPLC_MLP_Weights".w2[184] * v2[24] + "NeuroPLC_MLP_Weights".w2[185] * v2[25] + "NeuroPLC_MLP_Weights".w2[186] * v2[26] + "NeuroPLC_MLP_Weights".w2[187] * v2[27] + "NeuroPLC_MLP_Weights".w2[188] * v2[28] + "NeuroPLC_MLP_Weights".w2[189] * v2[29] + "NeuroPLC_MLP_Weights".w2[190] * v2[30] + "NeuroPLC_MLP_Weights".w2[191] * v2[31];
        v3[6] := "NeuroPLC_MLP_Weights".b3[6] + "NeuroPLC_MLP_Weights".w2[192] * v2[0] + "NeuroPLC_MLP_Weights".w2[193] * v2[1] + "NeuroPLC_MLP_Weights".w2[194] * v2[2] + "NeuroPLC_MLP_Weights".w2[195] * v2[3] + "NeuroPLC_MLP_Weights".w2[196] * v2[4] + "NeuroPLC_MLP_Weights".w2[197] * v2[5] + "NeuroPLC_MLP_Weights".w2[198] * v2[6] + "NeuroPLC_MLP_Weights".w2[199] * v2[7] + "NeuroPLC_MLP_Weights".w2[200] * v2[8] + "NeuroPLC_MLP_Weights".w2[201] * v2[9] + "NeuroPLC_MLP_Weights".w2[202] * v2[10] + "NeuroPLC_MLP_Weights".w2[203] * v2[11] + "NeuroPLC_MLP_Weights".w2[204] * v2[12] + "NeuroPLC_MLP_Weights".w2[205] * v2[13] + "NeuroPLC_MLP_Weights".w2[206] * v2[14] + "NeuroPLC_MLP_Weights".w2[207] * v2[15] + "NeuroPLC_MLP_Weights".w2[208] * v2[16] + "NeuroPLC_MLP_Weights".w2[209] * v2[17] + "NeuroPLC_MLP_Weights".w2[210] * v2[18] + "NeuroPLC_MLP_Weights".w2[211] * v2[19] + "NeuroPLC_MLP_Weights".w2[212] * v2[20] + "NeuroPLC_MLP_Weights".w2[213] * v2[21] + "NeuroPLC_MLP_Weights".w2[214] * v2[22] + "NeuroPLC_MLP_Weights".w2[215] * v2[23] + "NeuroPLC_MLP_Weights".w2[216] * v2[24] + "NeuroPLC_MLP_Weights".w2[217] * v2[25] + "NeuroPLC_MLP_Weights".w2[218] * v2[26] + "NeuroPLC_MLP_Weights".w2[219] * v2[27] + "NeuroPLC_MLP_Weights".w2[220] * v2[28] + "NeuroPLC_MLP_Weights".w2[221] * v2[29] + "NeuroPLC_MLP_Weights".w2[222] * v2[30] + "NeuroPLC_MLP_Weights".w2[223] * v2[31];
        v3[7] := "NeuroPLC_MLP_Weights".b3[7] + "NeuroPLC_MLP_Weights".w2[224] * v2[0] + "NeuroPLC_MLP_Weights".w2[225] * v2[1] + "NeuroPLC_MLP_Weights".w2[226] * v2[2] + "NeuroPLC_MLP_Weights".w2[227] * v2[3] + "NeuroPLC_MLP_Weights".w2[228] * v2[4] + "NeuroPLC_MLP_Weights".w2[229] * v2[5] + "NeuroPLC_MLP_Weights".w2[230] * v2[6] + "NeuroPLC_MLP_Weights".w2[231] * v2[7] + "NeuroPLC_MLP_Weights".w2[232] * v2[8] + "NeuroPLC_MLP_Weights".w2[233] * v2[9] + "NeuroPLC_MLP_Weights".w2[234] * v2[10] + "NeuroPLC_MLP_Weights".w2[235] * v2[11] + "NeuroPLC_MLP_Weights".w2[236] * v2[12] + "NeuroPLC_MLP_Weights".w2[237] * v2[13] + "NeuroPLC_MLP_Weights".w2[238] * v2[14] + "NeuroPLC_MLP_Weights".w2[239] * v2[15] + "NeuroPLC_MLP_Weights".w2[240] * v2[16] + "NeuroPLC_MLP_Weights".w2[241] * v2[17] + "NeuroPLC_MLP_Weights".w2[242] * v2[18] + "NeuroPLC_MLP_Weights".w2[243] * v2[19] + "NeuroPLC_MLP_Weights".w2[244] * v2[20] + "NeuroPLC_MLP_Weights".w2[245] * v2[21] + "NeuroPLC_MLP_Weights".w2[246] * v2[22] + "NeuroPLC_MLP_Weights".w2[247] * v2[23] + "NeuroPLC_MLP_Weights".w2[248] * v2[24] + "NeuroPLC_MLP_Weights".w2[249] * v2[25] + "NeuroPLC_MLP_Weights".w2[250] * v2[26] + "NeuroPLC_MLP_Weights".w2[251] * v2[27] + "NeuroPLC_MLP_Weights".w2[252] * v2[28] + "NeuroPLC_MLP_Weights".w2[253] * v2[29] + "NeuroPLC_MLP_Weights".w2[254] * v2[30] + "NeuroPLC_MLP_Weights".w2[255] * v2[31];
        v3[8] := "NeuroPLC_MLP_Weights".b3[8] + "NeuroPLC_MLP_Weights".w2[256] * v2[0] + "NeuroPLC_MLP_Weights".w2[257] * v2[1] + "NeuroPLC_MLP_Weights".w2[258] * v2[2] + "NeuroPLC_MLP_Weights".w2[259] * v2[3] + "NeuroPLC_MLP_Weights".w2[260] * v2[4] + "NeuroPLC_MLP_Weights".w2[261] * v2[5] + "NeuroPLC_MLP_Weights".w2[262] * v2[6] + "NeuroPLC_MLP_Weights".w2[263] * v2[7] + "NeuroPLC_MLP_Weights".w2[264] * v2[8] + "NeuroPLC_MLP_Weights".w2[265] * v2[9] + "NeuroPLC_MLP_Weights".w2[266] * v2[10] + "NeuroPLC_MLP_Weights".w2[267] * v2[11] + "NeuroPLC_MLP_Weights".w2[268] * v2[12] + "NeuroPLC_MLP_Weights".w2[269] * v2[13] + "NeuroPLC_MLP_Weights".w2[270] * v2[14] + "NeuroPLC_MLP_Weights".w2[271] * v2[15] + "NeuroPLC_MLP_Weights".w2[272] * v2[16] + "NeuroPLC_MLP_Weights".w2[273] * v2[17] + "NeuroPLC_MLP_Weights".w2[274] * v2[18] + "NeuroPLC_MLP_Weights".w2[275] * v2[19] + "NeuroPLC_MLP_Weights".w2[276] * v2[20] + "NeuroPLC_MLP_Weights".w2[277] * v2[21] + "NeuroPLC_MLP_Weights".w2[278] * v2[22] + "NeuroPLC_MLP_Weights".w2[279] * v2[23] + "NeuroPLC_MLP_Weights".w2[280] * v2[24] + "NeuroPLC_MLP_Weights".w2[281] * v2[25] + "NeuroPLC_MLP_Weights".w2[282] * v2[26] + "NeuroPLC_MLP_Weights".w2[283] * v2[27] + "NeuroPLC_MLP_Weights".w2[284] * v2[28] + "NeuroPLC_MLP_Weights".w2[285] * v2[29] + "NeuroPLC_MLP_Weights".w2[286] * v2[30] + "NeuroPLC_MLP_Weights".w2[287] * v2[31];
        v3[9] := "NeuroPLC_MLP_Weights".b3[9] + "NeuroPLC_MLP_Weights".w2[288] * v2[0] + "NeuroPLC_MLP_Weights".w2[289] * v2[1] + "NeuroPLC_MLP_Weights".w2[290] * v2[2] + "NeuroPLC_MLP_Weights".w2[291] * v2[3] + "NeuroPLC_MLP_Weights".w2[292] * v2[4] + "NeuroPLC_MLP_Weights".w2[293] * v2[5] + "NeuroPLC_MLP_Weights".w2[294] * v2[6] + "NeuroPLC_MLP_Weights".w2[295] * v2[7] + "NeuroPLC_MLP_Weights".w2[296] * v2[8] + "NeuroPLC_MLP_Weights".w2[297] * v2[9] + "NeuroPLC_MLP_Weights".w2[298] * v2[10] + "NeuroPLC_MLP_Weights".w2[299] * v2[11] + "NeuroPLC_MLP_Weights".w2[300] * v2[12] + "NeuroPLC_MLP_Weights".w2[301] * v2[13] + "NeuroPLC_MLP_Weights".w2[302] * v2[14] + "NeuroPLC_MLP_Weights".w2[303] * v2[15] + "NeuroPLC_MLP_Weights".w2[304] * v2[16] + "NeuroPLC_MLP_Weights".w2[305] * v2[17] + "NeuroPLC_MLP_Weights".w2[306] * v2[18] + "NeuroPLC_MLP_Weights".w2[307] * v2[19] + "NeuroPLC_MLP_Weights".w2[308] * v2[20] + "NeuroPLC_MLP_Weights".w2[309] * v2[21] + "NeuroPLC_MLP_Weights".w2[310] * v2[22] + "NeuroPLC_MLP_Weights".w2[311] * v2[23] + "NeuroPLC_MLP_Weights".w2[312] * v2[24] + "NeuroPLC_MLP_Weights".w2[313] * v2[25] + "NeuroPLC_MLP_Weights".w2[314] * v2[26] + "NeuroPLC_MLP_Weights".w2[315] * v2[27] + "NeuroPLC_MLP_Weights".w2[316] * v2[28] + "NeuroPLC_MLP_Weights".w2[317] * v2[29] + "NeuroPLC_MLP_Weights".w2[318] * v2[30] + "NeuroPLC_MLP_Weights".w2[319] * v2[31];
        v3[10] := "NeuroPLC_MLP_Weights".b3[10] + "NeuroPLC_MLP_Weights".w2[320] * v2[0] + "NeuroPLC_MLP_Weights".w2[321] * v2[1] + "NeuroPLC_MLP_Weights".w2[322] * v2[2] + "NeuroPLC_MLP_Weights".w2[323] * v2[3] + "NeuroPLC_MLP_Weights".w2[324] * v2[4] + "NeuroPLC_MLP_Weights".w2[325] * v2[5] + "NeuroPLC_MLP_Weights".w2[326] * v2[6] + "NeuroPLC_MLP_Weights".w2[327] * v2[7] + "NeuroPLC_MLP_Weights".w2[328] * v2[8] + "NeuroPLC_MLP_Weights".w2[329] * v2[9] + "NeuroPLC_MLP_Weights".w2[330] * v2[10] + "NeuroPLC_MLP_Weights".w2[331] * v2[11] + "NeuroPLC_MLP_Weights".w2[332] * v2[12] + "NeuroPLC_MLP_Weights".w2[333] * v2[13] + "NeuroPLC_MLP_Weights".w2[334] * v2[14] + "NeuroPLC_MLP_Weights".w2[335] * v2[15] + "NeuroPLC_MLP_Weights".w2[336] * v2[16] + "NeuroPLC_MLP_Weights".w2[337] * v2[17] + "NeuroPLC_MLP_Weights".w2[338] * v2[18] + "NeuroPLC_MLP_Weights".w2[339] * v2[19] + "NeuroPLC_MLP_Weights".w2[340] * v2[20] + "NeuroPLC_MLP_Weights".w2[341] * v2[21] + "NeuroPLC_MLP_Weights".w2[342] * v2[22] + "NeuroPLC_MLP_Weights".w2[343] * v2[23] + "NeuroPLC_MLP_Weights".w2[344] * v2[24] + "NeuroPLC_MLP_Weights".w2[345] * v2[25] + "NeuroPLC_MLP_Weights".w2[346] * v2[26] + "NeuroPLC_MLP_Weights".w2[347] * v2[27] + "NeuroPLC_MLP_Weights".w2[348] * v2[28] + "NeuroPLC_MLP_Weights".w2[349] * v2[29] + "NeuroPLC_MLP_Weights".w2[350] * v2[30] + "NeuroPLC_MLP_Weights".w2[351] * v2[31];
        v3[11] := "NeuroPLC_MLP_Weights".b3[11] + "NeuroPLC_MLP_Weights".w2[352] * v2[0] + "NeuroPLC_MLP_Weights".w2[353] * v2[1] + "NeuroPLC_MLP_Weights".w2[354] * v2[2] + "NeuroPLC_MLP_Weights".w2[355] * v2[3] + "NeuroPLC_MLP_Weights".w2[356] * v2[4] + "NeuroPLC_MLP_Weights".w2[357] * v2[5] + "NeuroPLC_MLP_Weights".w2[358] * v2[6] + "NeuroPLC_MLP_Weights".w2[359] * v2[7] + "NeuroPLC_MLP_Weights".w2[360] * v2[8] + "NeuroPLC_MLP_Weights".w2[361] * v2[9] + "NeuroPLC_MLP_Weights".w2[362] * v2[10] + "NeuroPLC_MLP_Weights".w2[363] * v2[11] + "NeuroPLC_MLP_Weights".w2[364] * v2[12] + "NeuroPLC_MLP_Weights".w2[365] * v2[13] + "NeuroPLC_MLP_Weights".w2[366] * v2[14] + "NeuroPLC_MLP_Weights".w2[367] * v2[15] + "NeuroPLC_MLP_Weights".w2[368] * v2[16] + "NeuroPLC_MLP_Weights".w2[369] * v2[17] + "NeuroPLC_MLP_Weights".w2[370] * v2[18] + "NeuroPLC_MLP_Weights".w2[371] * v2[19] + "NeuroPLC_MLP_Weights".w2[372] * v2[20] + "NeuroPLC_MLP_Weights".w2[373] * v2[21] + "NeuroPLC_MLP_Weights".w2[374] * v2[22] + "NeuroPLC_MLP_Weights".w2[375] * v2[23] + "NeuroPLC_MLP_Weights".w2[376] * v2[24] + "NeuroPLC_MLP_Weights".w2[377] * v2[25] + "NeuroPLC_MLP_Weights".w2[378] * v2[26] + "NeuroPLC_MLP_Weights".w2[379] * v2[27] + "NeuroPLC_MLP_Weights".w2[380] * v2[28] + "NeuroPLC_MLP_Weights".w2[381] * v2[29] + "NeuroPLC_MLP_Weights".w2[382] * v2[30] + "NeuroPLC_MLP_Weights".w2[383] * v2[31];
        v3[12] := "NeuroPLC_MLP_Weights".b3[12] + "NeuroPLC_MLP_Weights".w2[384] * v2[0] + "NeuroPLC_MLP_Weights".w2[385] * v2[1] + "NeuroPLC_MLP_Weights".w2[386] * v2[2] + "NeuroPLC_MLP_Weights".w2[387] * v2[3] + "NeuroPLC_MLP_Weights".w2[388] * v2[4] + "NeuroPLC_MLP_Weights".w2[389] * v2[5] + "NeuroPLC_MLP_Weights".w2[390] * v2[6] + "NeuroPLC_MLP_Weights".w2[391] * v2[7] + "NeuroPLC_MLP_Weights".w2[392] * v2[8] + "NeuroPLC_MLP_Weights".w2[393] * v2[9] + "NeuroPLC_MLP_Weights".w2[394] * v2[10] + "NeuroPLC_MLP_Weights".w2[395] * v2[11] + "NeuroPLC_MLP_Weights".w2[396] * v2[12] + "NeuroPLC_MLP_Weights".w2[397] * v2[13] + "NeuroPLC_MLP_Weights".w2[398] * v2[14] + "NeuroPLC_MLP_Weights".w2[399] * v2[15] + "NeuroPLC_MLP_Weights".w2[400] * v2[16] + "NeuroPLC_MLP_Weights".w2[401] * v2[17] + "NeuroPLC_MLP_Weights".w2[402] * v2[18] + "NeuroPLC_MLP_Weights".w2[403] * v2[19] + "NeuroPLC_MLP_Weights".w2[404] * v2[20] + "NeuroPLC_MLP_Weights".w2[405] * v2[21] + "NeuroPLC_MLP_Weights".w2[406] * v2[22] + "NeuroPLC_MLP_Weights".w2[407] * v2[23] + "NeuroPLC_MLP_Weights".w2[408] * v2[24] + "NeuroPLC_MLP_Weights".w2[409] * v2[25] + "NeuroPLC_MLP_Weights".w2[410] * v2[26] + "NeuroPLC_MLP_Weights".w2[411] * v2[27] + "NeuroPLC_MLP_Weights".w2[412] * v2[28] + "NeuroPLC_MLP_Weights".w2[413] * v2[29] + "NeuroPLC_MLP_Weights".w2[414] * v2[30] + "NeuroPLC_MLP_Weights".w2[415] * v2[31];
        v3[13] := "NeuroPLC_MLP_Weights".b3[13] + "NeuroPLC_MLP_Weights".w2[416] * v2[0] + "NeuroPLC_MLP_Weights".w2[417] * v2[1] + "NeuroPLC_MLP_Weights".w2[418] * v2[2] + "NeuroPLC_MLP_Weights".w2[419] * v2[3] + "NeuroPLC_MLP_Weights".w2[420] * v2[4] + "NeuroPLC_MLP_Weights".w2[421] * v2[5] + "NeuroPLC_MLP_Weights".w2[422] * v2[6] + "NeuroPLC_MLP_Weights".w2[423] * v2[7] + "NeuroPLC_MLP_Weights".w2[424] * v2[8] + "NeuroPLC_MLP_Weights".w2[425] * v2[9] + "NeuroPLC_MLP_Weights".w2[426] * v2[10] + "NeuroPLC_MLP_Weights".w2[427] * v2[11] + "NeuroPLC_MLP_Weights".w2[428] * v2[12] + "NeuroPLC_MLP_Weights".w2[429] * v2[13] + "NeuroPLC_MLP_Weights".w2[430] * v2[14] + "NeuroPLC_MLP_Weights".w2[431] * v2[15] + "NeuroPLC_MLP_Weights".w2[432] * v2[16] + "NeuroPLC_MLP_Weights".w2[433] * v2[17] + "NeuroPLC_MLP_Weights".w2[434] * v2[18] + "NeuroPLC_MLP_Weights".w2[435] * v2[19] + "NeuroPLC_MLP_Weights".w2[436] * v2[20] + "NeuroPLC_MLP_Weights".w2[437] * v2[21] + "NeuroPLC_MLP_Weights".w2[438] * v2[22] + "NeuroPLC_MLP_Weights".w2[439] * v2[23] + "NeuroPLC_MLP_Weights".w2[440] * v2[24] + "NeuroPLC_MLP_Weights".w2[441] * v2[25] + "NeuroPLC_MLP_Weights".w2[442] * v2[26] + "NeuroPLC_MLP_Weights".w2[443] * v2[27] + "NeuroPLC_MLP_Weights".w2[444] * v2[28] + "NeuroPLC_MLP_Weights".w2[445] * v2[29] + "NeuroPLC_MLP_Weights".w2[446] * v2[30] + "NeuroPLC_MLP_Weights".w2[447] * v2[31];
        v3[14] := "NeuroPLC_MLP_Weights".b3[14] + "NeuroPLC_MLP_Weights".w2[448] * v2[0] + "NeuroPLC_MLP_Weights".w2[449] * v2[1] + "NeuroPLC_MLP_Weights".w2[450] * v2[2] + "NeuroPLC_MLP_Weights".w2[451] * v2[3] + "NeuroPLC_MLP_Weights".w2[452] * v2[4] + "NeuroPLC_MLP_Weights".w2[453] * v2[5] + "NeuroPLC_MLP_Weights".w2[454] * v2[6] + "NeuroPLC_MLP_Weights".w2[455] * v2[7] + "NeuroPLC_MLP_Weights".w2[456] * v2[8] + "NeuroPLC_MLP_Weights".w2[457] * v2[9] + "NeuroPLC_MLP_Weights".w2[458] * v2[10] + "NeuroPLC_MLP_Weights".w2[459] * v2[11] + "NeuroPLC_MLP_Weights".w2[460] * v2[12] + "NeuroPLC_MLP_Weights".w2[461] * v2[13] + "NeuroPLC_MLP_Weights".w2[462] * v2[14] + "NeuroPLC_MLP_Weights".w2[463] * v2[15] + "NeuroPLC_MLP_Weights".w2[464] * v2[16] + "NeuroPLC_MLP_Weights".w2[465] * v2[17] + "NeuroPLC_MLP_Weights".w2[466] * v2[18] + "NeuroPLC_MLP_Weights".w2[467] * v2[19] + "NeuroPLC_MLP_Weights".w2[468] * v2[20] + "NeuroPLC_MLP_Weights".w2[469] * v2[21] + "NeuroPLC_MLP_Weights".w2[470] * v2[22] + "NeuroPLC_MLP_Weights".w2[471] * v2[23] + "NeuroPLC_MLP_Weights".w2[472] * v2[24] + "NeuroPLC_MLP_Weights".w2[473] * v2[25] + "NeuroPLC_MLP_Weights".w2[474] * v2[26] + "NeuroPLC_MLP_Weights".w2[475] * v2[27] + "NeuroPLC_MLP_Weights".w2[476] * v2[28] + "NeuroPLC_MLP_Weights".w2[477] * v2[29] + "NeuroPLC_MLP_Weights".w2[478] * v2[30] + "NeuroPLC_MLP_Weights".w2[479] * v2[31];
        v3[15] := "NeuroPLC_MLP_Weights".b3[15] + "NeuroPLC_MLP_Weights".w2[480] * v2[0] + "NeuroPLC_MLP_Weights".w2[481] * v2[1] + "NeuroPLC_MLP_Weights".w2[482] * v2[2] + "NeuroPLC_MLP_Weights".w2[483] * v2[3] + "NeuroPLC_MLP_Weights".w2[484] * v2[4] + "NeuroPLC_MLP_Weights".w2[485] * v2[5] + "NeuroPLC_MLP_Weights".w2[486] * v2[6] + "NeuroPLC_MLP_Weights".w2[487] * v2[7] + "NeuroPLC_MLP_Weights".w2[488] * v2[8] + "NeuroPLC_MLP_Weights".w2[489] * v2[9] + "NeuroPLC_MLP_Weights".w2[490] * v2[10] + "NeuroPLC_MLP_Weights".w2[491] * v2[11] + "NeuroPLC_MLP_Weights".w2[492] * v2[12] + "NeuroPLC_MLP_Weights".w2[493] * v2[13] + "NeuroPLC_MLP_Weights".w2[494] * v2[14] + "NeuroPLC_MLP_Weights".w2[495] * v2[15] + "NeuroPLC_MLP_Weights".w2[496] * v2[16] + "NeuroPLC_MLP_Weights".w2[497] * v2[17] + "NeuroPLC_MLP_Weights".w2[498] * v2[18] + "NeuroPLC_MLP_Weights".w2[499] * v2[19] + "NeuroPLC_MLP_Weights".w2[500] * v2[20] + "NeuroPLC_MLP_Weights".w2[501] * v2[21] + "NeuroPLC_MLP_Weights".w2[502] * v2[22] + "NeuroPLC_MLP_Weights".w2[503] * v2[23] + "NeuroPLC_MLP_Weights".w2[504] * v2[24] + "NeuroPLC_MLP_Weights".w2[505] * v2[25] + "NeuroPLC_MLP_Weights".w2[506] * v2[26] + "NeuroPLC_MLP_Weights".w2[507] * v2[27] + "NeuroPLC_MLP_Weights".w2[508] * v2[28] + "NeuroPLC_MLP_Weights".w2[509] * v2[29] + "NeuroPLC_MLP_Weights".w2[510] * v2[30] + "NeuroPLC_MLP_Weights".w2[511] * v2[31];

        // StandardAct: relu
        FOR i := 0 TO 15 DO
            IF v3[i] < 0.0 THEN
                v4[i] := 0.0;
            ELSE
                v4[i] := v3[i];
            END_IF;
        END_FOR;

        // MatMul: fc2
        v5[0] := "NeuroPLC_MLP_Weights".b5[0] + "NeuroPLC_MLP_Weights".w4[0] * v4[0] + "NeuroPLC_MLP_Weights".w4[1] * v4[1] + "NeuroPLC_MLP_Weights".w4[2] * v4[2] + "NeuroPLC_MLP_Weights".w4[3] * v4[3] + "NeuroPLC_MLP_Weights".w4[4] * v4[4] + "NeuroPLC_MLP_Weights".w4[5] * v4[5] + "NeuroPLC_MLP_Weights".w4[6] * v4[6] + "NeuroPLC_MLP_Weights".w4[7] * v4[7] + "NeuroPLC_MLP_Weights".w4[8] * v4[8] + "NeuroPLC_MLP_Weights".w4[9] * v4[9] + "NeuroPLC_MLP_Weights".w4[10] * v4[10] + "NeuroPLC_MLP_Weights".w4[11] * v4[11] + "NeuroPLC_MLP_Weights".w4[12] * v4[12] + "NeuroPLC_MLP_Weights".w4[13] * v4[13] + "NeuroPLC_MLP_Weights".w4[14] * v4[14] + "NeuroPLC_MLP_Weights".w4[15] * v4[15];
        v5[1] := "NeuroPLC_MLP_Weights".b5[1] + "NeuroPLC_MLP_Weights".w4[16] * v4[0] + "NeuroPLC_MLP_Weights".w4[17] * v4[1] + "NeuroPLC_MLP_Weights".w4[18] * v4[2] + "NeuroPLC_MLP_Weights".w4[19] * v4[3] + "NeuroPLC_MLP_Weights".w4[20] * v4[4] + "NeuroPLC_MLP_Weights".w4[21] * v4[5] + "NeuroPLC_MLP_Weights".w4[22] * v4[6] + "NeuroPLC_MLP_Weights".w4[23] * v4[7] + "NeuroPLC_MLP_Weights".w4[24] * v4[8] + "NeuroPLC_MLP_Weights".w4[25] * v4[9] + "NeuroPLC_MLP_Weights".w4[26] * v4[10] + "NeuroPLC_MLP_Weights".w4[27] * v4[11] + "NeuroPLC_MLP_Weights".w4[28] * v4[12] + "NeuroPLC_MLP_Weights".w4[29] * v4[13] + "NeuroPLC_MLP_Weights".w4[30] * v4[14] + "NeuroPLC_MLP_Weights".w4[31] * v4[15];
        v5[2] := "NeuroPLC_MLP_Weights".b5[2] + "NeuroPLC_MLP_Weights".w4[32] * v4[0] + "NeuroPLC_MLP_Weights".w4[33] * v4[1] + "NeuroPLC_MLP_Weights".w4[34] * v4[2] + "NeuroPLC_MLP_Weights".w4[35] * v4[3] + "NeuroPLC_MLP_Weights".w4[36] * v4[4] + "NeuroPLC_MLP_Weights".w4[37] * v4[5] + "NeuroPLC_MLP_Weights".w4[38] * v4[6] + "NeuroPLC_MLP_Weights".w4[39] * v4[7] + "NeuroPLC_MLP_Weights".w4[40] * v4[8] + "NeuroPLC_MLP_Weights".w4[41] * v4[9] + "NeuroPLC_MLP_Weights".w4[42] * v4[10] + "NeuroPLC_MLP_Weights".w4[43] * v4[11] + "NeuroPLC_MLP_Weights".w4[44] * v4[12] + "NeuroPLC_MLP_Weights".w4[45] * v4[13] + "NeuroPLC_MLP_Weights".w4[46] * v4[14] + "NeuroPLC_MLP_Weights".w4[47] * v4[15];
        v5[3] := "NeuroPLC_MLP_Weights".b5[3] + "NeuroPLC_MLP_Weights".w4[48] * v4[0] + "NeuroPLC_MLP_Weights".w4[49] * v4[1] + "NeuroPLC_MLP_Weights".w4[50] * v4[2] + "NeuroPLC_MLP_Weights".w4[51] * v4[3] + "NeuroPLC_MLP_Weights".w4[52] * v4[4] + "NeuroPLC_MLP_Weights".w4[53] * v4[5] + "NeuroPLC_MLP_Weights".w4[54] * v4[6] + "NeuroPLC_MLP_Weights".w4[55] * v4[7] + "NeuroPLC_MLP_Weights".w4[56] * v4[8] + "NeuroPLC_MLP_Weights".w4[57] * v4[9] + "NeuroPLC_MLP_Weights".w4[58] * v4[10] + "NeuroPLC_MLP_Weights".w4[59] * v4[11] + "NeuroPLC_MLP_Weights".w4[60] * v4[12] + "NeuroPLC_MLP_Weights".w4[61] * v4[13] + "NeuroPLC_MLP_Weights".w4[62] * v4[14] + "NeuroPLC_MLP_Weights".w4[63] * v4[15];

        // Softmax
        max_val := v5[0];
        FOR i := 1 TO 3 DO
            IF v5[i] > max_val THEN
                max_val := v5[i];
            END_IF;
        END_FOR;
        sum := 0.0;
        FOR i := 0 TO 3 DO
            v6[i] := EXP(v5[i] - max_val);
            sum := sum + v6[i];
        END_FOR;
        FOR i := 0 TO 3 DO
            v6[i] := v6[i] / sum;
        END_FOR;

        // Argmax
        max_val := v6[0];
        fault_class := 0;
        FOR i := 1 TO 3 DO
            IF v6[i] > max_val THEN
                max_val := v6[i];
                fault_class := i;
            END_IF;
        END_FOR;
        confidence := max_val;

END_FUNCTION_BLOCK
